(* IEC 61131-3 sources: beebread/doc (part 5) *)

(* ---- beedance_network.st ---- *)
// Commented out for beedance: it uses _STRING_TO_BUFFER, which is commented out.
// FUNCTION_BLOCK BASE64_DECODE_STR
// VAR_INPUT
// 	RUN : BOOL;
// END_VAR
// VAR_OUTPUT
// 	DONE : BOOL;
// END_VAR
// VAR_IN_OUT
// 	STR1 : STRING(192);
// 	STR2 : STRING(144);
// END_VAR
// VAR
// 	BASE64_DECODE_STREAM : BASE64_DECODE_STREAM;
// 	run_last : BOOL;
// 	buf1 : ARRAY [0..63] OF BYTE;
// 	buf2 : ARRAY [0..47] OF BYTE;
// 	mode : INT;
// 	size1 : INT;
// 	size2 : INT;
// 	end : INT;
// 	pos : INT;
// END_VAR
//
// CASE mode OF
// 0:	IF RUN AND NOT run_last THEN
// 		DONE := FALSE;
// 		mode := 1;
// 		end := LEN(STR1);
// 		pos := 0;
// 		STR2 := '';
// 	END_IF;
// 1:
// 	size1 := MIN(48,end - pos);
// 	IF size1 > 0 THEN
// 		_STRING_TO_BUFFER(STR:=MID(STR1, size1, pos + 1), POS:=0, PT:=REF(buf1), SIZE:=SIZEOF(buf1));
// 		BASE64_DECODE_STREAM(BUF1:=buf1 ,BUF2:=buf2 ,SIZE1:=size1 ,SIZE2=>size2);
// 		STR2 := CONCAT(STR2,BUFFER_TO_STRING(PT:=REF(buf2), SIZE:=SIZEOF(buf2), START:=0, STOP:=size2 - 1));
// 	ELSE
// 		mode := 0;
// 		DONE := TRUE;
// 	END_IF;
// 	pos := pos + size1;
// END_CASE;
//
// run_last := RUN;
// END_FUNCTION_BLOCK

FUNCTION_BLOCK BASE64_DECODE_STREAM
VAR_IN_OUT
	BUF1 : ARRAY [0..63] OF BYTE;
	BUF2 : ARRAY [0..47] OF BYTE;
END_VAR
VAR_INPUT
	SIZE1 : INT;
END_VAR
VAR_OUTPUT
	SIZE2 : INT;
END_VAR
VAR_TEMP
	a: INT;
	b: WORD;
	o: INT;
	off: INT;
	i1: INT;
	i2: INT;
	c: INT;
END_VAR

IF SIZE1 <= 0 THEN SIZE2 := 0; RETURN; END_IF;
c := SIZE1 - 1;
i2 := 0;
a := 0;
b := 0;
FOR i1 := 0 TO c DO
	o := BUF1[i1];
	IF o = 61 THEN (* = *)	EXIT;
	ELSIF o > 96 THEN (* a-z *) off := 71;
	ELSIF o > 64 THEN (* A-Z *) off := 65;
	ELSIF o > 47 THEN (* 0-9 *) off := -4;
	ELSIF o = 43 THEN (* + *) off := -19;
	ELSIF o = 47 THEN (* / *) off := -16;
	END_IF;
	b := SHL(b,6) OR INT_TO_BYTE(o - off);
	a := a + 6;
	IF a >= 8 THEN
		a := a - 8;
		BUF2[i2] := WORD_TO_BYTE(SHR(b,a));
		i2 := i2 + 1;
		b := b AND NOT SHL(WORD#16#FFFF,a);
	END_IF;
END_FOR;
SIZE2 := i2;
END_FUNCTION_BLOCK

// Commented out for beedance: it uses _STRING_TO_BUFFER, which is commented out.
// FUNCTION_BLOCK BASE64_ENCODE_STR
// VAR_INPUT
// 	RUN : BOOL;
// END_VAR
// VAR_OUTPUT
// 	DONE : BOOL;
// END_VAR
// VAR_IN_OUT
// 	STR1 : STRING(144);
// 	STR2 : STRING(192);
// END_VAR
// VAR
// 	BASE64_ENCODE_STREAM : BASE64_ENCODE_STREAM;
// 	run_last : BOOL;
// 	buf1 : ARRAY [0..47] OF BYTE;
// 	buf2 : ARRAY [0..63] OF BYTE;
// 	mode : INT;
// 	size1 : INT;
// 	size2 : INT;
// 	end : INT;
// 	pos : INT;
// END_VAR
//
// CASE mode OF
// 0:	IF RUN AND NOT run_last THEN
// 		DONE := FALSE;
// 		mode := 1;
// 		end := LEN(STR1);
// 		pos := 0;
// 		STR2 := '';
// 	END_IF;
// 1:
// 	size1 := MIN(48,end - pos);
// 	IF size1 > 0 THEN
// 		_STRING_TO_BUFFER(STR:=MID(STR1, size1, pos + 1), POS:=0, PT:=REF(buf1), SIZE:=SIZEOF(buf1));
// 		BASE64_ENCODE_STREAM(BUF1:=buf1 ,BUF2:=buf2 ,SIZE1:=size1 ,SIZE2=>size2);
// 		STR2 := CONCAT(STR2,BUFFER_TO_STRING(PT:=REF(buf2), SIZE:=SIZEOF(buf2), START:=0, STOP:=size2 - 1));
// 	ELSE
// 		mode := 0;
// 		DONE := TRUE;
// 	END_IF;
// 	pos := pos + size1;
// END_CASE;
//
// run_last := RUN;
// END_FUNCTION_BLOCK

// Commented out for beedance: it uses CODE, which is commented out.
// FUNCTION_BLOCK BASE64_ENCODE_STREAM
// VAR_IN_OUT
// 	BUF1 : ARRAY [0..47] OF BYTE;
// 	BUF2 : ARRAY [0..63] OF BYTE;
// END_VAR
// VAR_INPUT
// 	SIZE1 : INT;
// END_VAR
// VAR_OUTPUT
// 	SIZE2 : INT;
// END_VAR
// VAR
// 	a: INT;
// 	b: WORD;
// 	i: INT;
// 	i2: INT;
// 	i3: INT;
// 	c: INT;
// 	BASE64: STRING(64) := 'ABCDEFGHIJKLMNOPQRSTUVWXYZabcdefghijklmnopqrstuvwxyz0123456789+/';
// END_VAR
//
// IF SIZE1 <= 0 THEN
// 	SIZE2 := 0;
// 	RETURN;
// END_IF;
// c := SIZE1 - 1;
// i2 := 0;
// a := 0;
// b := 0;
// FOR i := 0 TO c DO
// 	b := SHL(b,8) OR BUF1[i];
// 	a := a + 8;
// 	WHILE a >= 6 DO
// 		a := a - 6;
// 		buf2[i2] := CODE(BASE64,WORD_TO_INT(SHR(b,a)) + 1);
// 		i2 := i2 + 1;
// 		b := b AND NOT SHL(WORD#16#FFFF,a);
// 	END_WHILE;
// END_FOR;
// IF a > 0 THEN
// 	buf2[i2] := CODE(BASE64,WORD_TO_INT(SHL(b,6 - a)) + 1);
// 	i2 := i2 + 1;
// 	i3 := i2 + (NOT INT_TO_WORD(i2) AND 2#11);
// 	FOR i := i2 TO i3 DO
// 		buf2[i] := 61;
// 	END_FOR;
// 	SIZE2 := i3 + 1;
// ELSE
// 	SIZE2 := i2;
// END_IF;
// END_FUNCTION_BLOCK

// Commented out for beedance: it reads or writes the bytes of a STRING through a pointer; a beedance reference (REF_TO) refers to a whole variable of its type.
// FUNCTION_BLOCK CSV_PARSER_BUF
// VAR_INPUT
// 	SEP : BYTE;
// END_VAR
// VAR_IN_OUT
// 	RUN : BYTE;
// 	OFFSET : UDINT;
// 	VALUE : STRING(STRING_LENGTH);
// 	PT : NETWORK_BUFFER;
// END_VAR
// VAR_OUTPUT
// 	RESULT : BYTE;
// END_VAR
// VAR
// 	step : INT;
// 	size : INT;
// 	c : BYTE;
// 	v_add : BYTE;
// 	i : INT;
// 	state : BYTE;
// 	eof : BOOL;
// 	pv : REF_TO BYTE;
// 	pve : DWORD;
// 	watchdog : TON;
// 	x : BOOL;
//
// 	(*LOG_MSG : LOG_MSG;
// 	_debug_enable : BOOL := TRUE;
// 	step_last : INT;*)
// END_VAR
//
// IF RUN > 0 THEN
// 	IF state = 0 THEN (* restart evaluation *)
//
// 		pv := REF(VALUE);
// 		pv^ := 0; (* VALUE = '' *)
// 		pve := pv + INT_TO_DWORD(STRING_LENGTH);
// 		i := UDINT_TO_INT(OFFSET);
// 		size := UINT_TO_INT(PT.SIZE) - 1;
// 		RESULT := 0;
// 		state := 5; (* command in progress (busy) *)
// 		step := 0; (* restart evaluation *)
//
// 		(* ---------------- Debug-Message -----------------------*)
// 		(*IF _debug_enable THEN
// 			LOG_CL.NEW_MSG := 'CPF: Startindex: ~1';
// 			LOG_CL.PRINTF[1] := INT_TO_STRING(i);
// 			LOG_MSG();
// 		END_IF;*)
// 		(* -----------------------------------------------------------------*)
//
// 	END_IF;
//
// 	watchdog(IN:=FALSE,PT:=T#1ms); (* restart timer *)
// 	watchdog.IN := TRUE;
//
// 	WHILE (state = 5) DO (* loop as long as there is no result *)
//
// 		watchdog(); (* update timer *)
//
// 		IF watchdog.Q THEN (* watchdog triggered *)
// 			state := 5;
// 			EXIT;
// 		ELSIF i > size THEN (* no further character available *)
// 			state := 10; (* nothing found - end of data reached *)
// 			EXIT;
// 		ELSE
//
// 			c := PT.BUFFER[i]; (* read new character from buffer *)
// 			eof := i + 1 = PT.SIZE; (* End of File *)
//
// 			v_add := 0;
//
// 			IF c = SEP THEN (* new element detected *)
// 				state := 1;
// 				x := TRUE;
// 			ELSIF c >= 32 THEN (* element detected *)
// 				v_add := c; (* store character *)
// 				IF eof THEN
// 					state := 2; (* element and end of line detected *)
// 				ELSE
// 					x := TRUE;
// 				END_IF;
// 			ELSE
// 				IF x THEN
// 					state := 2; (* element and end of line detected *)
// 					x := FALSE;
// 				END_IF;
// 			END_IF;
//
// 			IF v_add > 0  AND pv < pve THEN (* add character to value string *)
// 				pv^ := v_add; (* enter character *)
// 				pv := pv + 1;
// 				pv^ := 0; (* enter string termination *)
// 			END_IF;
//
// 			i := i + 1; (* increment data pointer *)
//
// 		END_IF;
// 	END_WHILE;
//
// 	CASE state OF
// 	01:	(* element found *)
// 		RESULT := 1; (* element found *)
// 		OFFSET := i; (* take offset *)
// 		RUN := 0;
// 		state := 0;
// 	02:	(* element found *)
// 		RESULT := 2; (* element and end of line detected *)
// 		OFFSET := i; (* take offset *)
// 		RUN := 0;
// 		state := 0;
//
// 	05:	RESULT := 5; (* in progress *)
//
// 	10:	(* index out of range - end of buffer *)
// 		RESULT := 10; (* nothing found - end of data reached *)
// 		OFFSET := i; (* take offset *)
// 		RUN := 0;
// 		state := 0;
// 	END_CASE;
//
// 	(* ---------------- Debug-Message -----------------------*)
// 	(*IF _debug_enable THEN
// 		LOG_CL.NEW_MSG := 'CPF: intern Result ~1 , state ~2, step ~3 , offset ~4, run ~5';
// 		LOG_CL.PRINTF[1] := BYTE_TO_STRING(RESULT);
// 		LOG_CL.PRINTF[2] := BYTE_TO_STRING(state);
// 		LOG_CL.PRINTF[3] := INT_TO_STRING(step);
// 		LOG_CL.PRINTF[4] := UDINT_TO_STRING(OFFSET);
// 		LOG_CL.PRINTF[5] := BYTE_TO_STRING(RUN);
// 		LOG_MSG();
// 	END_IF;*)
// 	(* -----------------------------------------------------------------*)
//
// END_IF;
//
// (* ---------------- Debug-Message -----------------------*)
// (*IF _debug_enable THEN
// 	IF step_last <> step THEN
// 		LOG_CL.NEW_MSG := 'IPB: Step: ~1';
// 		LOG_CL.PRINTF[1]  := INT_TO_STRING(step);
// 		LOG_MSG();
// 	END_IF;
// 	step_last := step;
// END_IF;*)
// (* -----------------------------------------------------------------*)
// END_FUNCTION_BLOCK

// Commented out for beedance: it reads or writes the bytes of a STRING through a pointer; a beedance reference (REF_TO) refers to a whole variable of its type.
// FUNCTION_BLOCK CSV_PARSER_FILE
// VAR_INPUT
// 	SEP : BYTE;
// END_VAR
// VAR_IN_OUT
// 	FILENAME : STRING;
// 	FSD : FILE_SERVER_DATA;
// 	RUN : BYTE;
// 	OFFSET : UDINT;
// 	VALUE : STRING(STRING_LENGTH);
// 	PT	: NETWORK_BUFFER;
// END_VAR
// VAR_OUTPUT
// 	RESULT : BYTE;
// END_VAR
// VAR
// 	i : UDINT;
// 	state : BYTE;
// 	e : BYTE;
// 	mode : BYTE;
// 	step : INT;
// 	c : BYTE;
// 	v_add : BYTE;
// 	eof : BOOL;
// 	pv : REF_TO BYTE;
// 	pve : DWORD;
// 	watchdog : TON;
// 	x : BOOL;
// 	FB : FILE_BLOCK;
//
// 	(*LOG_MSG : LOG_MSG;
// 	_debug_enable : BOOL := FALSE;
// 	step_last : INT;*)
// END_VAR
//
// IF RUN > 0 THEN
//
// 	IF state = 0 THEN (* restart evaluation *)
// 		pv := REF(VALUE);
// 		pv^ := 0; (* VALUE = '' *)
// 		pve := pv + INT_TO_DWORD(STRING_LENGTH);
// 		i := OFFSET;
// 		RESULT := 0;
// 		state := 5; (* command in progress (busy) *)
// 		step := 0; (* restart evaluation *)
//
// 		(* ---------------- Debug-Message -----------------------*)
// 		(*IF _debug_enable THEN
// 			LOG_CL.NEW_MSG := 'CPF: Startindex: ~1';
// 			LOG_CL.PRINTF[1] := UDINT_TO_STRING(i);
// 			LOG_MSG();
// 		END_IF;*)
// 		(* -----------------------------------------------------------------*)
//
// 	END_IF;
//
// 	watchdog(IN:=FALSE,PT:=T#1ms); (* restart timer *)
// 	watchdog.IN := TRUE;
//
// 	WHILE (state = 5) DO (* loop as long as there is no result *)
//
// 		mode := 1;
// 		FB(MODE:=mode,FSD:=fsd,PT:=PT,FILENAME:=FILENAME,POS:=i );
// 		e:=FB.ERROR;
// 		c:=FB.DATA;
//
// 		eof := i + 1 = FSD.FILE_SIZE; (* End of File *)
//
// 		(* ---------------- Debug-Message -----------------------*)
// 		(*IF _debug_enable THEN
// 			LOG_CL.NEW_MSG := 'CPF: mode: ~1, error: ~2 , >~7<>~3< ~4 step ~5 index ~6';
// 			LOG_CL.PRINTF[1] := BYTE_TO_STRING(mode);
// 			LOG_CL.PRINTF[2] := BYTE_TO_STRING(e);
// 			LOG_CL.PRINTF[3] := BYTE_TO_STRING(c);
// 			LOG_CL.PRINTF[4] := BOOL_TO_STRING(eof);
// 			LOG_CL.PRINTF[5] := INT_TO_STRING(step);
// 			LOG_CL.PRINTF[6] := UDINT_TO_STRING(i);
// 			LOG_CL.PRINTF[7] := CHR_TO_STRING(c);
// 			LOG_MSG();
// 		END_IF;*)
// 		(* -----------------------------------------------------------------*)
// 		watchdog(); (* update timer *)
//
// 		IF mode > 0 OR watchdog.Q THEN (* block still active, or watchdog triggered *)
// 			state := 5;
// 			EXIT;
// 		ELSIF e > 0 THEN (* File_error or no further character available *)
// 			state := 10; (* nothing found - end of data reached *)
// 			EXIT;
// 		ELSE
//
// 			v_add := 0;
//
// 			IF c = SEP THEN (* new element detected *)
// 				state := 1;
// 				x := TRUE;
// 			ELSIF c >= 32 THEN (* element detected *)
// 				v_add := c; (* store character *)
// 				IF eof THEN
// 					state := 2; (* element and end of line detected *)
// 				ELSE
// 					x := TRUE;
// 				END_IF;
// 			ELSE
// 				IF x THEN
// 					state := 2; (* element and end of line detected *)
// 					x := FALSE;
// 				END_IF;
// 			END_IF;
//
// 			IF v_add > 0  AND pv < pve THEN (* add character to value string *)
// 				pv^ := v_add; (* enter character *)
// 				pv := pv + 1;
// 				pv^ := 0; (* enter string termination *)
// 			END_IF;
//
// 			i := i + 1; (* increment data pointer *)
//
// 		END_IF;
// 	END_WHILE;
//
// 	CASE state OF
// 	01:	(* element found *)
// 		RESULT := 1; (* element found *)
// 		OFFSET := i; (* take offset *)
// 		RUN := 0;
// 		state := 0;
// 	02:	(* element found *)
// 		RESULT := 2; (* element and end of line detected *)
// 		OFFSET := i; (* take offset *)
// 		RUN := 0;
// 		state := 0;
//
// 	05:	RESULT := 5; (* in progress *)
//
// 	10:	(* index out of range - end of buffer *)
// 		RESULT := 10; (* nothing found - end of data reached *)
// 		OFFSET := i; (* take offset *)
// 		RUN := 0;
// 		state := 0;
// 	END_CASE;
//
// 	(* ---------------- Debug-Message -----------------------*)
// 	(*IF _debug_enable THEN
// 		LOG_CL.NEW_MSG := 'CPF: intern Result ~1 , state ~2, step ~3 , offset ~4, run ~5';
// 		LOG_CL.PRINTF[1] := BYTE_TO_STRING(RESULT);
// 		LOG_CL.PRINTF[2] := BYTE_TO_STRING(state);
// 		LOG_CL.PRINTF[3] := INT_TO_STRING(step);
// 		LOG_CL.PRINTF[4] := UDINT_TO_STRING(OFFSET);
// 		LOG_CL.PRINTF[5] := BYTE_TO_STRING(RUN);
// 		LOG_MSG();
// 	END_IF;*)
// 	(* -----------------------------------------------------------------*)
//
// END_IF;
//
// (* ---------------- Debug-Message -----------------------*)
// (*IF _debug_enable THEN
// 	IF step_last <> step THEN
// 		LOG_CL.NEW_MSG := 'CPF: Step: ~1';
// 		LOG_CL.PRINTF[1]  := INT_TO_STRING(step);
// 		LOG_MSG();
// 	END_IF;
// 	step_last := step;
// END_IF;*)
// (* -----------------------------------------------------------------*)
// END_FUNCTION_BLOCK

// Commented out for beedance: it uses UNI_CIRCULAR_BUFFER, which is commented out.
// FUNCTION_BLOCK DLOG_BOOL
// VAR_IN_OUT
// 	X : DLOG_DATA;
// END_VAR
// VAR_INPUT
// 	STATE : BOOL;
// 	OFF : STRING;
// 	ON : STRING;
// 	COLUMN : STRING(40);
// 	DELTA : BOOL;
// END_VAR
// VAR_OUTPUT
// END_VAR
// VAR
// 	UCB : UNI_CIRCULAR_BUFFER;
// 	id : WORD;
// 	last_delta : BOOL;
// 	state_last: BOOL;
// END_VAR
//
// CASE x.ADD_COM OF
//
// 01:	(* ADD INFO *)
// 	X.ID_MAX := X.ID_MAX + USINT#1;
// 	id := WORD#16#0601; (* source type BOOL, target type STRING *)
// 02:	(* ADD HEADER *)
// 	X.UCB.D_STRING := COLUMN;
// 	X.UCB.D_HEAD := id;
// 	X.UCB.D_MODE := 1;
// 	UCB(DATA:=X.UCB); (* enter data *)
// 03:	(* ADD DATA *)
// 	IF X.STORE_TYPE = BYTE#05 THEN (* MySQL mode *)
// 		X.UCB.D_STRING := SEL(state_last,'0','1');
// 	ELSE
// 		X.UCB.D_STRING := SEL(state_last,OFF,ON);
// 	END_IF;
// 	X.UCB.D_HEAD := id;
//
// 	X.UCB.D_MODE := 1;
// 	UCB(DATA:=X.UCB); (* enter data *)
// 	last_delta := STATE;
// 04:	(* ADD DATA REQ *)
// 	IF DELTA AND (STATE XOR last_delta) THEN
// 		X.ADD_DATA_REQ := TRUE;
// 		last_delta := STATE;
// 	END_IF;
// END_CASE;
// state_last := STATE;
// END_FUNCTION_BLOCK

// Commented out for beedance: it uses ELEMENT_GET, which is commented out.
// FUNCTION_BLOCK DLOG_CRON_TAB
// VAR_INPUT
// 	ACTIVATE : BOOL;
// 	DTI : DT;
// 	SECOND : STRING(20);
// 	MINUTE : STRING(20);
// 	HOUR : STRING(20);
// 	DAY_OF_MONTH : STRING(20);
// 	DAY_OF_WEEK : STRING(20);
// 	MONTH : STRING(20);
// END_VAR
// VAR_OUTPUT
// 	Q : BOOL;
// END_VAR
// VAR
// 	CD :  DLOG_CRON_DATA;
// 	activate_old : BOOL;
// 	datei : DATE;
// 	dti_last : DT;
// 	cnt1 : INT;
// 	cnt2 : INT;
// 	idx1 : INT;
// 	idx2 : INT;
// 	idx3 : INT;
// 	idx4 : INT;
// 	pos1 : INT;
// 	pos2 : INT;
// 	char_cnt : INT;
// 	trig_day : BOOL;
// 	trig_weekday : BOOL;
// 	str1 : STRING(STRING_LENGTH);
// 	str2 : STRING(STRING_LENGTH);
// 	str3 : STRING(STRING_LENGTH);
// 	num_str1 : STRING(10);
// END_VAR
//
// IF ACTIVATE THEN
// 	IF NOT activate_old THEN
// 		CD.CE[0].VALUE_MIN := 0;	(* seconds *)
// 		CD.CE[0].VALUE_MAX := 59;
// 		CD.CE[1].VALUE_MIN := 0;	(* minutes *)
// 		CD.CE[1].VALUE_MAX := 59;
// 		CD.CE[2].VALUE_MIN := 0;	(* hours *)
// 		CD.CE[2].VALUE_MAX := 59;
// 		CD.CE[3].VALUE_MIN := 1;	(* days *)
// 		CD.CE[3].VALUE_MAX := 31;
// 		CD.CE[4].VALUE_MIN := 1;	(* weekday *)
// 		CD.CE[4].VALUE_MAX := 7;
// 		CD.CE[5].VALUE_MIN := 1;	(* month *)
// 		CD.CE[5].VALUE_MAX := 12;
//
// 		FOR idx1 := 0 TO 5 DO
// 			idx3 := CD.CE[idx1].VALUE_MIN;
// 			idx4 := CD.CE[idx1].VALUE_MAx;
// 			FOR idx2 := idx3 TO idx4 DO
// 				CD.CE[idx1].ELEMENTS[idx2] := FALSE;
// 			END_FOR;
// 			CD.CE[idx1].ALL_SELECTED := FALSE;
// 		END_FOR;
//
// 		str1 := CONCAT(SECOND,'#');
// 		str1 := CONCAT(str1,MINUTE);
// 		str1 := CONCAT(str1,'#');
// 		str1 := CONCAT(str1,HOUR);
// 		str1 := CONCAT(str1,'#');
// 		str1 := CONCAT(str1,DAY_OF_MONTH);
// 		str1 := CONCAT(str1,'#');
// 		str1 := CONCAT(str1,DAY_OF_WEEK);
// 		str1 := CONCAT(str1,'#');
// 		str1 := CONCAT(str1,MONTH);
//
// 		FOR idx1 := 0 TO 5 DO
// 			str2 := ELEMENT_GET(BYTE#35, idx1, str1);
// 			IF LEN(str2) > 0 THEN
// 				cnt1 := ELEMENT_COUNT(BYTE#44, str2);	(* separator ',' *)
// 			ELSE
// 				cnt1 := 1;
// 			END_IF;
//
// 			FOR idx2 := 0 TO cnt1 -1 DO
// 				str3 := ELEMENT_GET(BYTE#44, idx2, str2);
// 				IF FIND(str3, '*/') > 0 AND LEN(str3) <= 10 THEN
// 					pos1 := DEC_TO_INT(str3);
// 					IF pos1 > 0 THEN
// 						idx3 := CD.CE[idx1].VALUE_MIN;
// 						idx4 := CD.CE[idx1].VALUE_MAX;
// 						WHILE idx3 <= idx4 DO
// 							CD.CE[idx1].ELEMENTS[idx3] := TRUE;
// 							idx3 := idx3 + pos1;
// 						END_WHILE;
// 					END_IF;
//
// 				ELSE
// 					IF FIND(str3, '*') > 0 OR LEN(str3) = 0 THEN
// 						pos1 := CD.CE[idx1].VALUE_MIN;
// 						pos2 := CD.CE[idx1].VALUE_MAX;
// 						CD.CE[idx1].ALL_SELECTED := TRUE;
// 					ELSE
// 						cnt2 := ELEMENT_COUNT(BYTE#45, str3);	(* separator '-' *)
// 						char_cnt := LEN(str3);
// 						IF char_cnt >= 1 AND char_cnt <= 10 THEN
// 							num_str1 := ELEMENT_GET(BYTE#45, 0, str3);
// 							pos1 := DEC_TO_INT(num_str1);
// 							pos2 := pos1;
// 							IF cnt2 = 2 THEN
// 								num_str1 := ELEMENT_GET(BYTE#45, 1, str3);
// 								pos2 := DEC_TO_INT(num_str1);
// 							END_IF;
// 						END_IF;
// 					END_IF;
//
// 					IF pos1 >= CD.CE[idx1].VALUE_MIN AND pos2 <= CD.CE[idx1].VALUE_MAX THEN
// 						FOR idx3 := pos1 TO pos2 DO
// 							CD.CE[idx1].ELEMENTS[idx3] := TRUE;
// 						END_FOR;
// 					END_IF;
// 				END_IF;
// 			END_FOR;
// 		END_FOR;
// 	ELSIF DTI <> dti_last THEN
// 		CD.CE[0].VALUE := SECOND_OF_DT(DTI); (* seconds *)
// 		CD.CE[1].VALUE := MINUTE_OF_DT(DTI); (* minutes *)
// 		CD.CE[2].VALUE := HOUR_OF_DT(DTI); (* hours *)
// 		datei := DT_TO_DATE(DTI);
// 		CD.CE[3].VALUE := DAY_OF_MONTH(datei); (* Tag *)
// 		CD.CE[4].VALUE := DAY_OF_WEEK(datei); (* weekday *)
// 		CD.CE[5].VALUE := MONTH_OF_DATE(datei); (*  month *)
// 		dti_last := DTI;
//
// 		idx2 := CD.CE[0].VALUE;	(* seconds *)
// 		Q := CD.CE[0].ELEMENTS[idx2] = TRUE;
// 		idx2 := CD.CE[1].VALUE;	(* minutes *)
// 		Q := Q AND CD.CE[1].ELEMENTS[idx2] = TRUE;
// 		idx2 := CD.CE[2].VALUE;	(* hours *)
// 		Q := Q AND CD.CE[2].ELEMENTS[idx2] = TRUE;
// 		idx2 := CD.CE[5].VALUE;	(* month *)
// 		Q := Q AND CD.CE[5].ELEMENTS[idx2] = TRUE;
//
// 		(* evaluate day and weekday *)
// 		idx2 := CD.CE[3].VALUE;	(* Tag *)
// 		trig_day:= CD.CE[3].ELEMENTS[idx2] = TRUE;
// 		idx2 := CD.CE[4].VALUE;	(* weekday *)
// 		trig_weekday := CD.CE[4].ELEMENTS[idx2] = TRUE;
//
// 		IF CD.CE[3].ALL_SELECTED = FALSE AND CD.CE[4].ALL_SELECTED = TRUE THEN
// 			Q := Q AND trig_day; (* evaluate day only *)
// 		ELSIF CD.CE[3].ALL_SELECTED = TRUE AND CD.CE[4].ALL_SELECTED = FALSE THEN
// 			Q := Q AND trig_weekday; (* evaluate weekday only *)
// 		ELSIF CD.CE[3].ALL_SELECTED = FALSE AND CD.CE[4].ALL_SELECTED = FALSE THEN
// 			Q := Q AND (trig_weekday OR trig_day); (* evaluate day and weekday *)
// 		END_IF;
// 	END_IF;
//
// END_IF;
// activate_old := ACTIVATE;
// END_FUNCTION_BLOCK

// Commented out for beedance: it uses UNI_CIRCULAR_BUFFER, which is commented out.
// FUNCTION_BLOCK DLOG_DINT
// VAR_IN_OUT
// 	X : DLOG_DATA;
// END_VAR
// VAR_INPUT
// 	VALUE : DINT;
// 	COLUMN : STRING(40);
// 	DELTA : DINT;
// END_VAR
// VAR
// 	UCB : UNI_CIRCULAR_BUFFER;
// 	id : WORD;
// 	delta_last : DINT;
// 	value_last : DINT;
// END_VAR
//
// CASE x.ADD_COM OF
//
// 01:	(* ADD INFO *)
// 	X.ID_MAX := X.ID_MAX + USINT#1;
// 	id := WORD#16#0801; (* source type DINT, target type STRING *)
// 02:	(* ADD HEADER *)
// 	X.UCB.D_STRING := COLUMN;
// 	X.UCB.D_HEAD := id;
// 	X.UCB.D_MODE := 1;
// 	UCB(DATA:=X.UCB); (* enter data *)
// 03:	(* ADD DATA *)
// 	X.UCB.D_STRING := DINT_TO_STRING(value_last);
// 	X.UCB.D_HEAD := id;
// 	X.UCB.D_MODE := 1;
// 	UCB(DATA:=X.UCB); (* enter data *)
// 	delta_last := value_last;
// 04:	(* ADD DATA REQ *)
// 	IF DELTA <> DINT#0 THEN
// 		IF VALUE <= (delta_last - DELTA) OR VALUE >= (delta_last + DELTA) THEN
// 			X.ADD_DATA_REQ := TRUE;
// 			delta_last := VALUE;
// 		END_IF;
// 	END_IF;
// END_CASE;
// value_last := VALUE;
// END_FUNCTION_BLOCK

// Commented out for beedance: it uses UNI_CIRCULAR_BUFFER, which is commented out.
// FUNCTION_BLOCK DLOG_DT
// VAR_IN_OUT
// 	X : DLOG_DATA;
// END_VAR
// VAR_INPUT
// 	FMT : STRING := '#A-#D-#H #N:#R:#T';
// 	COLUMN : STRING(40);
// 	DELTA : UDINT;
// END_VAR
//
// VAR_OUTPUT
// END_VAR
// VAR
// 	UCB : UNI_CIRCULAR_BUFFER;
// 	id : WORD;
// 	delta_last : DT;
// END_VAR
//
// CASE x.ADD_COM OF
//
// 01:	(* ADD INFO *)
// 	X.ID_MAX := X.ID_MAX + USINT#1;
// 	id := WORD#16#0D01; (* source type DT, target type STRING *)
// 02:	(* ADD HEADER *)
// 	X.UCB.D_STRING := COLUMN;
// 	X.UCB.D_HEAD := id;
// 	X.UCB.D_MODE := 1;
// 	UCB(DATA:=X.UCB); (* enter data *)
// 03:	(* ADD DATA *)
// 	X.UCB.D_STRING := DT_TO_STRF(DTI:=X.DTI,MS:=0,FMT:=FMT,LANG:=0);
// 	X.UCB.D_HEAD := id;
// 	X.UCB.D_MODE := 1;
// 	UCB(DATA:=X.UCB); (* enter data *)
// 	delta_last := X.DTI;
// 04:	(* ADD DATA REQ *)
// 	IF DELTA <> UDINT#0 THEN
// 		IF DT_TO_UDINT(X.DTI) >= (DT_TO_UDINT(delta_last) + DELTA) THEN
// 			X.ADD_DATA_REQ := TRUE;
// 			delta_last := X.DTI;
// 		END_IF;
// 	END_IF;
// END_CASE;
// END_FUNCTION_BLOCK

// Commented out for beedance: it uses UNI_CIRCULAR_BUFFER, which is commented out.
// FUNCTION_BLOCK DLOG_FILE_TO_FTP
// VAR_IN_OUT
// 	X : DLOG_DATA;
// END_VAR
// VAR_INPUT
// 	FTP_URL : STRING(STRING_LENGTH);
// 	FTP_ACTIV : BOOL;
// 	FILE_DELETE : BOOL;
// 	TIMEOUT : TIME := T#30s;
// 	RETRY : INT;
// 	RETRY_TIME : TIME := T#30s;
// 	DNS_IP4 : DWORD;
// 	PLC_IP4 : DWORD;
// END_VAR
// VAR_OUTPUT
// 	DONE : BOOL;
// 	BUSY : BOOL;
// 	ERROR_C : DWORD;
// 	ERROR_T : BYTE;
// END_VAR
// VAR
// 	UCBD : UNI_CIRCULAR_BUFFER_DATA;
// 	UCB : UNI_CIRCULAR_BUFFER;
// 	FTP_CLIENT : FTP_CLIENT;
// 	WT_1 : TON;
// 	ftrig_old : BOOL;
// 	filename : STRING;
// 	step : INT;
// 	ftp_busy : BOOL;
// 	ftp_done : BOOL;
// 	cnt : INT;
//
// 	(*LOG_MSG : LOG_MSG;
// 	_debug_enable : BOOL := TRUE;*)
// END_VAR
//
// (* store new file name *)
// IF X.NEW_FILE_RTRIG AND ftrig_old = FALSE THEN
// 	UCBD.D_HEAD := 1;
// 	UCBD.D_MODE := 1;
// 	UCBD.D_STRING := X.NEW_FILE;
// 	UCB(DATA:=UCBD); (* enter data *)
// END_IF;
// ftrig_old := X.NEW_FILE_RTRIG;
//
// CASE step OF
//
// 00:	IF UCBD.BUF_COUNT > 0 AND ftp_busy = FALSE THEN
// 		UCBD.D_MODE := 12; (* read and delete data *)
// 		UCB(DATA:=UCBD);
// 		filename := UCBD.D_STRING;
// 		cnt := RETRY;
// 		step := 10;
//
// 		(*####################  DEBUG-MESSAGE  ###################################*)
// 		(*IF _debug_enable THEN
// 			LOG_CL.NEW_MSG := 'F_T_FTP: Auftrag aktiv /file: ~2';
// 			LOG_CL.PRINTF[2] := files;
// 			LOG_MSG();
// 		END_IF;*)
// 		(*########################################################################*)
//
// 	END_IF;
//
// 10:	IF ftp_busy = FALSE THEN
// 		IF ftp_done THEN
// 			(*####################  DEBUG-MESSAGE  ###################################*)
// 			(*IF _debug_enable THEN
// 				LOG_CL.NEW_MSG := 'F_T_FTP: Auftrag OK /file: ~2';
// 				LOG_CL.PRINTF[2] := filename;
// 				LOG_MSG();
// 			END_IF;*)
// 			(*########################################################################*)
// 			step := 0;
// 		ELSE
// 			step := 20; (* pause after error *)
// 		END_IF;
// 	END_IF;
//
// 20:	IF WT_1.Q THEN (* wait time *)
// 		cnt := cnt - 1;
// 		IF RETRY = 0 THEN (* repeat FTP transfer indefinitely *)
// 			(*####################  DEBUG-MESSAGE  ###################################*)
// 			(*IF _debug_enable THEN
// 				LOG_CL.NEW_MSG := 'F_T_FTP: Auftrag unbegrenzt wiederholen /file: ~2';
// 				LOG_CL.PRINTF[2] := filename;
// 				LOG_MSG();
// 			END_IF;*)
// 			(*########################################################################*)
// 			step := 10; (* repeat FTP transfer *)
// 		ELSIF cnt >= 0 THEN
// 			(*####################  DEBUG-MESSAGE  ###################################*)
// 			(*IF _debug_enable THEN
// 				LOG_CL.NEW_MSG := 'F_T_FTP: Auftrag wiederholen /cnt: ~1 /file: ~2';
// 				LOG_CL.PRINTF[1] := INT_TO_STRING(cnt);
// 				LOG_CL.PRINTF[2] := filename;
// 				LOG_MSG();
// 			END_IF;*)
// 			(*########################################################################*)
// 			step := 10; (* repeat FTP transfer *)
// 		ELSE
// 			(*####################  DEBUG-MESSAGE  ###################################*)
// 			(*IF _debug_enable THEN
// 				LOG_CL.NEW_MSG := 'F_T_FTP: Auftrag verworfen /file: ~2';
// 				LOG_CL.PRINTF[2] := filename;
// 				LOG_MSG();
// 			END_IF;*)
// 			(*########################################################################*)
// 			step := 0; (* discard FTP job *)
// 		END_IF;
// 	END_IF;
//
// END_CASE;
//
// BUSY := step = 10;
// DONE := step = 0;
// WT_1(IN:= step = 20, PT:= RETRY_TIME);
//
// FTP_CLIENT(
// 	ACTIVATE:= BUSY,
// 	FILENAME:= filename,
// 	FTP_URL:= FTP_URL,
// 	FTP_DOWNLOAD:= FALSE,
// 	FTP_ACTIV:= FTP_ACTIV,
// 	FILE_DELETE:= FILE_DELETE,
// 	TIMEOUT:= TIMEOUT,
// 	DNS_IP4:= DNS_IP4,
// 	PLC_IP4:= PLC_IP4,
// 	DONE=> ftp_done,
// 	BUSY=> ftp_busy
// 	);
//
// (* error evaluation *)
// IF FTP_CLIENT.ERROR_T <> BYTE#0 THEN
// 	ERROR_C := FTP_CLIENT.ERROR_C;
// 	ERROR_T := FTP_CLIENT.ERROR_T;
// ELSIF UCBD.BUF_DATA_LOST > UDINT#0 THEN
// 	ERROR_C := DWORD#2; (* error: buffer overflow - reduce amount of data *)
// 	ERROR_T := BYTE#6; 	(* Type: Buffer *)
// ELSIF UCBD.BUF_USED_MAX > USINT#90 THEN
// 	ERROR_C := DWORD#1; (* warning: buffer utilization > 90% *)
// 	ERROR_T := BYTE#6;	(* Type: Buffer *)
// ELSE
// 	ERROR_C := DWORD#0;
// 	ERROR_T := BYTE#0;
// END_IF;
// END_FUNCTION_BLOCK

// Commented out for beedance: it uses UNI_CIRCULAR_BUFFER, which is commented out.
// FUNCTION_BLOCK DLOG_FILE_TO_SMTP
// VAR_IN_OUT
// 	SERVER : STRING;
// 	MAILFROM : STRING;
// 	MAILTO : STRING(STRING_LENGTH);
// 	SUBJECT : STRING;
// 	BODY : STRING(STRING_LENGTH);
// 	X : DLOG_DATA;
// END_VAR
// VAR_INPUT
// 	FILE_DELETE : BOOL;
// 	TIMEOUT : TIME := T#30s;
// 	DTI : DT;
// 	DTI_OFFSET : INT;
// 	RETRY : INT;
// 	RETRY_TIME : TIME := T#30s;
// 	DNS_IP4 : DWORD;
// END_VAR
// VAR_OUTPUT
// 	DONE : BOOL;
// 	BUSY : BOOL;
// 	ERROR_C : DWORD;
// 	ERROR_T : BYTE;
// END_VAR
// VAR
// 	UCBD : UNI_CIRCULAR_BUFFER_DATA;
// 	UCB : UNI_CIRCULAR_BUFFER;
// 	SMTP_CLIENT : SMTP_CLIENT;
// 	WT_1 : TON;
// 	ftrig_old : BOOL;
// 	files : STRING(STRING_LENGTH);
// 	step : INT;
// 	smtp_busy : BOOL;
// 	smtp_done : BOOL;
// 	cnt : INT;
//
// 	(*LOG_MSG : LOG_MSG;
// 	_debug_enable : BOOL := TRUE;*)
// END_VAR
//
// (* store new file name *)
// IF X.NEW_FILE_RTRIG AND ftrig_old = FALSE THEN
// 	UCBD.D_HEAD := 1;
// 	UCBD.D_MODE := 1;
// 	UCBD.D_STRING := X.NEW_FILE;
// 	UCB(DATA:=UCBD); (* enter data *)
// END_IF;
// ftrig_old := X.NEW_FILE_RTRIG;
//
// CASE step OF
//
// 00:	IF UCBD.BUF_COUNT > 0 AND smtp_busy = FALSE THEN
// 		UCBD.D_MODE := 12; (* read and delete data *)
// 		UCB(DATA:=UCBD);
// 		files := UCBD.D_STRING;
// 		IF FILE_DELETE THEN
// 			files := CONCAT(files,';#DEL#');
// 		END_IF;
// 		cnt := RETRY;
// 		step := 10;
//
// 		(*####################  DEBUG-MESSAGE  ###################################*)
// 		(*IF _debug_enable THEN
// 			LOG_CL.NEW_MSG := 'F_T_SMTP: Auftrag aktiv /file: ~2';
// 			LOG_CL.PRINTF[2] := files;
// 			LOG_MSG();
// 		END_IF;*)
// 		(*########################################################################*)
//
// 	END_IF;
//
// 10:	IF smtp_busy = FALSE THEN
// 		IF smtp_done THEN
// 			(*####################  DEBUG-MESSAGE  ###################################*)
// 			(*IF _debug_enable THEN
// 				LOG_CL.NEW_MSG := 'F_T_SMTP: Auftrag OK /file: ~2';
// 				LOG_CL.PRINTF[2] := files;
// 				LOG_MSG();
// 			END_IF;*)
// 			(*########################################################################*)
// 			step := 0;
// 		ELSE
// 			step := 20; (* pause after error *)
// 		END_IF;
// 	END_IF;
//
// 20:	IF WT_1.Q THEN (* wait time *)
// 		cnt := cnt - 1;
// 		IF RETRY = 0 THEN (* repeat transfer indefinitely *)
// 			(*####################  DEBUG-MESSAGE  ###################################*)
// 			(*IF _debug_enable THEN
// 				LOG_CL.NEW_MSG := 'F_T_SMTP: Auftrag unbegrenzt wiederholen /file: ~2';
// 				LOG_CL.PRINTF[2] := files;
// 				LOG_MSG();
// 			END_IF;*)
// 			(*########################################################################*)
// 			step := 10; (* repeat transfer *)
// 		ELSIF cnt >= 0 THEN
// 			(*####################  DEBUG-MESSAGE  ###################################*)
// 			(*IF _debug_enable THEN
// 				LOG_CL.NEW_MSG := 'F_T_SMTP: Auftrag wiederholen /cnt: ~1 /file: ~2';
// 				LOG_CL.PRINTF[1] := INT_TO_STRING(cnt);
// 				LOG_CL.PRINTF[2] := files;
// 				LOG_MSG();
// 			END_IF;*)
// 			(*########################################################################*)
// 			step := 10; (* repeat transfer *)
// 		ELSE
// 			(*####################  DEBUG-MESSAGE  ###################################*)
// 			(*IF _debug_enable THEN
// 				LOG_CL.NEW_MSG := 'F_T_SMTP: Auftrag verworfen /file: ~2';
// 				LOG_CL.PRINTF[2] := files;
// 				LOG_MSG();
// 			END_IF;*)
// 			(*########################################################################*)
// 			step := 0; (* discard job *)
// 		END_IF;
// 	END_IF;
//
// END_CASE;
//
// BUSY := step = 10;
// DONE := step = 0;
// WT_1(IN:= step = 20, PT:= RETRY_TIME);
//
// SMTP_CLIENT(
// 	ACTIVATE:= BUSY,
// 	TIMEOUT:= TIMEOUT,
// 	DTI:= DTI,
// 	DTI_OFFSET:= DTI_OFFSET,
// 	DNS_IP4:= DNS_IP4,
// 	SERVER:= SERVER,
// 	MAILFROM:= MAILFROM,
// 	MAILTO:= MAILTO,
// 	SUBJECT:= SUBJECT,
// 	BODY:= BODY,
// 	FILES:= FILES,
// 	DONE=> smtp_done,
// 	BUSY=> smtp_busy
// 	);
//
// (* error evaluation *)
// IF SMTP_CLIENT.ERROR_T <> BYTE#0 THEN
// 	ERROR_C := SMTP_CLIENT.ERROR_C;
// 	ERROR_T := SMTP_CLIENT.ERROR_T;
// ELSIF UCBD.BUF_DATA_LOST > UDINT#0 THEN
// 	ERROR_C := DWORD#2; (* error: buffer overflow - reduce amount of data *)
// 	ERROR_T := BYTE#6; 	(* Type: Buffer *)
// ELSIF UCBD.BUF_USED_MAX > USINT#90 THEN
// 	ERROR_C := DWORD#1; (* warning: buffer utilization > 90% *)
// 	ERROR_T := BYTE#6;	(* Type: Buffer *)
// ELSE
// 	ERROR_C := DWORD#0;
// 	ERROR_T := BYTE#0;
// END_IF;
// END_FUNCTION_BLOCK

// Commented out for beedance: it uses UNI_CIRCULAR_BUFFER, which is commented out.
// FUNCTION_BLOCK DLOG_REAL
// VAR_IN_OUT
// 	X : DLOG_DATA;
// END_VAR
// VAR_INPUT
// 	VALUE : REAL;
// 	N : INT;
// 	D : STRING(1) := ',';
// 	COLUMN : STRING(40);
// 	DELTA : REAL;
// END_VAR
// VAR
// 	UCB : UNI_CIRCULAR_BUFFER;
// 	id : WORD;
// 	delta_last : REAL;
// 	value_last : REAL;
// END_VAR
//
// CASE x.ADD_COM OF
//
// 01:	(* ADD INFO *)
// 	X.ID_MAX := X.ID_MAX + USINT#1;
// 	id := WORD#16#0201; (* source type REAL, target type STRING *)
// 02:	(* ADD HEADER *)
// 	X.UCB.D_STRING := COLUMN;
// 	X.UCB.D_HEAD := id;
// 	X.UCB.D_MODE := 1;
// 	UCB(DATA:=X.UCB); (* enter data *)
// 03:	(* ADD DATA *)
// 	X.UCB.D_STRING := REAL_TO_STRF(IN:=value_last,N:=N,D:=D);
// 	X.UCB.D_HEAD := id;
// 	X.UCB.D_MODE := 1;
// 	UCB(DATA:=X.UCB); (* enter data *)
// 	delta_last := value_last;
// 04:	(* ADD DATA REQ *)
// 	IF DELTA <> 0.0 THEN
// 		IF VALUE <= (delta_last - DELTA) OR VALUE >= (delta_last + DELTA) THEN
// 			X.ADD_DATA_REQ := TRUE;
// 			delta_last := VALUE;
// 		END_IF;
// 	END_IF;
// END_CASE;
// value_last := VALUE;
// END_FUNCTION_BLOCK

// Commented out for beedance: it uses UNI_CIRCULAR_BUFFER, which is commented out.
// FUNCTION_BLOCK DLOG_REAL_ARRAY
// VAR_IN_OUT
// 	R_ARRAY : DLOG_REAL_ARRAY_DATA;
// 	X : DLOG_DATA;
// END_VAR
// VAR_INPUT
// 	N : INT;
// 	D : STRING(1);
// 	R_COUNT : INT;
// END_VAR
// VAR
// 	UCB : UNI_CIRCULAR_BUFFER;
// 	id : WORD;
// 	idx : INT;
// END_VAR
//
// FOR idx := 1 TO R_COUNT DO
//
// 	CASE x.ADD_COM OF
//
// 	01:	(* ADD INFO *)
// 		X.ID_MAX := X.ID_MAX + USINT#1;
// 		id := WORD#16#0201; (* source type REAL, target type STRING *)
// 		(* assign name automatically *)
// 		IF LEN(R_ARRAY[idx].COLUMN) = 0 THEN
// 			R_ARRAY[idx].COLUMN := CONCAT('Spalte_',USINT_TO_STRING(X.ID_MAX));
// 		END_IF;
// 	02:	(* ADD HEADER *)
// 		X.UCB.D_STRING := R_ARRAY[idx].COLUMN;
// 		X.UCB.D_HEAD := id;
// 		X.UCB.D_MODE := 1;
// 		UCB(DATA:=X.UCB); (* enter data *)
// 	03:	(* ADD DATA *)
// 		X.UCB.D_STRING := REAL_TO_STRF(IN:=R_ARRAY[idx]._value_last,N:=N,D:=D);
// 		X.UCB.D_HEAD := id;
// 		X.UCB.D_MODE := 1;
// 		UCB(DATA:=X.UCB); (* enter data *)
// 		R_ARRAY[idx]._delta_last := R_ARRAY[idx]._value_last;
// 	04:	(* ADD DATA REQ *)
// 		IF R_ARRAY[idx].DELTA <> 0.0 THEN
// 			IF R_ARRAY[idx].VALUE <= (R_ARRAY[idx]._delta_last - R_ARRAY[idx].DELTA) OR R_ARRAY[idx].VALUE >= (R_ARRAY[idx]._delta_last + R_ARRAY[idx].DELTA) THEN
// 				X.ADD_DATA_REQ := TRUE;
// 				R_ARRAY[idx]._delta_last := R_ARRAY[idx].VALUE;
// 			END_IF;
// 		END_IF;
// 	END_CASE;
// 	R_ARRAY[idx]._value_last := R_ARRAY[idx].VALUE;
//
// END_FOR;
// END_FUNCTION_BLOCK

// Commented out for beedance: it names a variable fn, which beedance reads as its function keyword.
// FUNCTION_BLOCK DLOG_STORE_FILE_CSV
// VAR_IN_OUT
// 	X : DLOG_DATA;
// 	SAVE_DATA : DLOG_SAVE;
// END_VAR
// VAR_INPUT
// 	ENABLE : BOOL;
// 	TRIG_M : BOOL;
// 	TRIG_T : TIME;
// 	FILENAME : STRING;
// 	DTI : DT;
// 	SEP : BYTE;
// 	AUTO_CLOSE : TIME := T#15s;
// END_VAR
// VAR_OUTPUT
// 	ERROR_C : DWORD;
// 	ERROR_T : BYTE;
// END_VAR
// VAR
// 	FS : FILE_SERVER;
// 	FSD : FILE_SERVER_DATA;
// 	PT : NETWORK_BUFFER;
// 	UCB : UNI_CIRCULAR_BUFFER;
// 	trig_auto : BOOL;
// 	trig_stored : BOOL;
// 	trig_tmp : BOOL;
// 	trig_m_last : BOOL;
// 	dti_last : DT := DT#2070-02-06-06:28:15;
// 	fn_last : STRING;
// 	fn : STRING;
// 	step_1: INT;
// 	step_2: INT;
// 	idx : INT;
// 	log_stop : BOOL;
// 	n : USINT;
// 	wd_ton : TON;
// 	wd_time : TIME;
// 	aw_ton : TON;
// 	aw_enable : BOOL;
// 	aw_aktiv : BOOL;
// 	total_bytes : UDINT;
//
// 	(*
// 	LOG_MSG : LOG_MSG;
// 	_debug_enable : BOOL := TRUE;
// 	*)
// END_VAR
//
// X.DTI := DTI; (* enter date / time *)
// X.CLOCK_TRIG := DTI <> dti_last;
// dti_last := DTI;
// trig_auto := FALSE;
// IF X.CLOCK_TRIG THEN (* pulse every second *)
// 	fn := DT_TO_STRF(DTI, 0, FILENAME, 0); (* automatic file name generation *)
// 	IF TRIG_T >= T#1000ms THEN (* automatic trigger *)
// 		trig_auto := DT_TO_UDINT(DTI) MOD (TIME_TO_UDINT(TRIG_T) / UDINT#1000) = UDINT#0;
// 	END_IF;
// END_IF;
//
// CASE step_1 OF
//
// 00:	IF ENABLE THEN
// 		aw_enable := AUTO_CLOSE >= T#5s;
// 		wd_time := SEL(X.LOAD_TIME_MAX > T#0s, T#5ms,X.LOAD_TIME_MAX);
// 		fn_last := fn; (* store current file name *)
// 		IF X.ID_MAX = USINT#0 THEN (* scan for satellite blocks only once *)
// 			X.ADD_COM := 01; (* ADD INFO *)
// 			X.STORE_TYPE := BYTE#2; (* CSV mode *)
// 		END_IF;
// 		step_1 := 10;
//
// 		(* ---------------- Debug-Message -----------------------*)
// 		(*IF _debug_enable THEN
// 			LOG_CL.NEW_MSG := 'FILE_CSV1 - Start: File [~1], [~2]';
// 			LOG_CL.PRINTF[1] := fn_last;
// 			LOG_CL.PRINTF[2] := DT_TO_STRING(DTI);
// 			LOG_MSG();
// 		END_IF;*)
// 		(* -----------------------------------------------------------------*)
//
// 	END_IF;
//
// 10:	X.UCB.D_STRING := fn_last;
// 	IF fn_last = SAVE_DATA.FN_REM THEN
// 		X.UCB.D_HEAD := WORD#16#F201; (* Filemode open + write *)
// 		X.ADD_COM := 00;
// 	ELSE
// 		X.UCB.D_HEAD := WORD#16#F301; (* Filemode create + write *)
// 		X.ADD_COM := 02; (* ADD HEADER *)
// 	END_IF;
//
// 	X.UCB.D_MODE := 1; (* store file name as string *)
// 	UCB(DATA:=X.UCB); (* enter data *)
// 	step_1 := 30;
//
// 30:	(* process LOG trigger *)
// 	trig_tmp := (TRIG_M AND NOT trig_m_last) OR trig_auto OR X.ADD_DATA_REQ;
//
// 	IF ENABLE = FALSE OR fn <> fn_last THEN (* ENABLE = 0 or new file name -> log stop *)
// 		trig_stored := trig_tmp; (* store current trigger pulse *)
// 		X.UCB.D_HEAD := WORD#16#EE00;
// 		X.UCB.D_MODE := 1;
// 		UCB(DATA:=X.UCB); (* write element *)
// 		X.ADD_COM := 00;
// 		step_1 := 00;
//
// 		(* ---------------- Debug-Message -----------------------*)
// 		(*IF _debug_enable THEN
// 			LOG_CL.NEW_MSG := 'FILE_CSV1 - Stop: [~2]';
// 			LOG_CL.PRINTF[2] := DT_TO_STRING(DTI);
// 			LOG_MSG();
// 		END_IF;*)
// 		(* -----------------------------------------------------------------*)
//
// 	ELSIF ENABLE THEN
// 		IF trig_tmp OR trig_stored THEN (* manual, automatic or external trigger *)
// 			trig_stored := FALSE;
// 			X.ADD_COM := 03; (* ADD DATA *)
// 			SAVE_DATA.TRIG_CNT := SAVE_DATA.TRIG_CNT + UDINT#1;
// 			SAVE_DATA.TRIG_CNT_TOTAL  := SAVE_DATA.TRIG_CNT_TOTAL + UDINT#1;
// 			(* ---------------- Debug-Message -----------------------*)
// 			(*IF _debug_enable THEN
// 				LOG_CL.NEW_MSG := 'FILE_CSV1 - Trig: [~2]';
// 				LOG_CL.PRINTF[2] := DT_TO_STRING(DTI);
// 				LOG_MSG();
// 			END_IF;*)
// 			(* -----------------------------------------------------------------*)
// 		ELSE
// 			X.ADD_COM := 04;	(* ADD DATA REQ *)
// 		END_IF;
// 	END_IF;
//
// END_CASE;
// X.ADD_DATA_REQ := FALSE; (* reset external request *)
//
// (* ##################################### *)
//
// CASE step_2 OF
//
// 00:	aw_ton(IN:= idx > 0 AND aw_enable, PT:= AUTO_CLOSE); (* AutoWrite Timer *)
// 	IF aw_ton.Q THEN (* time-controlled data writing *)
// 		aw_aktiv := TRUE;
// 		step_2 := 10; (* write data *)
// 		(* ---------------- Debug-Message -----------------------*)
// 		(*IF _debug_enable THEN
// 			LOG_CL.NEW_MSG := 'FILE_CSV2 - AutoWrite: [~2]';
// 			LOG_CL.PRINTF[2] := DT_TO_STRING(DTI);
// 			LOG_MSG();
// 		END_IF;*)
// 		(* -----------------------------------------------------------------*)
//
// 	ELSE
// 		wd_ton(IN:= FALSE, PT:= wd_time);
// 		wd_ton(IN:= TRUE);
// 		WHILE X.UCB.BUF_COUNT > 0 AND step_2 = 0 AND wd_ton.Q = FALSE DO
//
// 			X.UCB.D_MODE := 10;
// 			UCB(DATA:=X.UCB); (* read element, but do not remove it yet *)
// 			IF X.UCB.D_HEAD > WORD#16#F000 THEN (* F301 or F201 *)
// 				X.UCB.D_MODE := 11;
// 				UCB(DATA:=X.UCB); (* remove element *)
//
// 				FSD.MODE := WORD_TO_BYTE(SHR(SHL(X.UCB.D_HEAD,4),12)); (* 0X00 -> 000X = 3 create + write / 2 open + write *)
// 				FSD.OFFSET := UDINT#0; (* start at beginning of file *)
// 				FSD.FILENAME := X.UCB.D_STRING; (* file name *)
// 				PT.SIZE := UINT#0;
// 				SAVE_DATA.FN_REM := FSD.FILENAME; (* save current file name as retained *)
//
// 				IF FSD.MODE = BYTE#3 THEN	(* create new file -> then reset counter *)
// 					SAVE_DATA.TRIG_CNT := UDINT#0;
// 				END_IF;
//
// 				X.NEW_FILE := FSD.FILENAME;
// 				X.NEW_FILE_SIZE := UDINT#0;
// 				X.NEW_FILE_RTRIG := FALSE;
// 				step_2 := 20;
// 				(* ---------------- Debug-Message -----------------------*)
// 				(*IF _debug_enable THEN
// 					LOG_CL.NEW_MSG := 'FILE_CSV2 - Create: Mode [~1] , [~2]';
// 					LOG_CL.PRINTF[2] := DT_TO_STRING(DTI);
// 					LOG_CL.PRINTF[1] := BYTE_TO_STRING(FSD.MODE);
// 					LOG_MSG();
// 				END_IF;*)
// 				(* -----------------------------------------------------------------*)
//
// 			ELSIF X.UCB.D_HEAD = WORD#16#EE00 THEN (* LOG_STOP Command *)
// 				X.UCB.D_MODE := 11;
// 				UCB(DATA:=X.UCB); (* remove element *)
// 				log_stop := TRUE;
// 				step_2 := 10; (* write data *)
//
// 			ELSIF idx + X.UCB.D_SIZE + 2 < SIZEOF(PT.BUFFER) THEN (* buffer space available *)
// 				X.UCB.D_MODE := 11;
// 				UCB(DATA:=X.UCB); (* remove element *)
// 				(* ---------------- Debug-Message -----------------------*)
// 				(*IF _debug_enable THEN
// 					LOG_CL.NEW_MSG := 'FILE_CSV2 - BUF: TXT [~1],Pos [~2], [~3]';
// 					LOG_CL.PRINTF[1] := X.UCB.D_STRING;
// 					LOG_CL.PRINTF[2] := INT_TO_STRING(idx);
// 					LOG_CL.PRINTF[3] := DT_TO_STRING(DTI);
// 					LOG_MSG();
// 				END_IF;*)
// 				(* -----------------------------------------------------------------*)
// 				_STRING_TO_BUFFER(STR:=X.UCB.D_STRING, POS:=idx, PT:=REF(PT.BUFFER), SIZE:=SIZEOF(PT.BUFFER));
// 				idx := idx + LEN(X.UCB.D_STRING);
// 				n := n + USINT#1;
// 				IF n = X.ID_MAX THEN (* last element of a line *)
// 					n := USINT#0;
// 					PT.BUFFER[idx] := BYTE#16#0D;
// 					idx := idx + 1;
// 					PT.BUFFER[idx] := BYTE#16#0A;
// 				ELSE
// 					PT.BUFFER[idx] := SEP;
// 				END_IF;
// 				idx := idx + 1;
// 				X.NEW_FILE_SIZE := total_bytes + INT_TO_UDINT(idx);
// 			ELSE (* no space available *)
// 				step_2 := 10; (* write data *)
// 			END_IF;
// 			wd_ton();
// 		END_WHILE;
// 	END_IF;
//
// 10:	IF idx > 0 THEN (* write data *)
// 		FSD.MODE := BYTE#2; (* File_Open_Exist + File_Write *)
// 		FSD.OFFSET := UDINT#4294967294; (* 16#FFFF_FFFE -> special code: automatically append data to end of file *)
// 		PT.SIZE := INT_TO_UINT(idx); (* enter data length *)
// 		idx := 0;
// 		(* ---------------- Debug-Message -----------------------*)
// 		(*IF _debug_enable THEN
// 			LOG_CL.NEW_MSG := 'FILE_CSV2 - WriteData: Mode [~3] Size [~1] , [~2]';
// 			LOG_CL.PRINTF[1] := UINT_TO_STRING(PT.SIZE);
// 			LOG_CL.PRINTF[2] := DT_TO_STRING(DTI);
// 			LOG_CL.PRINTF[3] := BYTE_TO_STRING(FSD.MODE);
// 			LOG_MSG();
// 		END_IF;*)
// 		(* -----------------------------------------------------------------*)
// 	END_IF;
// 	step_2 := 20;
//
// 20:	IF FSD.MODE = BYTE#0 THEN
// 		total_bytes := FSD.FILE_SIZE;
// 		X.NEW_FILE_SIZE := total_bytes + INT_TO_UDINT(idx);
// 		IF log_stop OR aw_aktiv THEN
// 			aw_aktiv := FALSE;
// 			FSD.MODE := BYTE#5; (* close file *)
// 			(* ---------------- Debug-Message -----------------------*)
// 			(*IF _debug_enable THEN
// 				LOG_CL.NEW_MSG := 'FILE_CSV2 - Close: [~2]';
// 				LOG_CL.PRINTF[2] := DT_TO_STRING(DTI);
// 				LOG_MSG();
// 			END_IF;*)
// 			(* -----------------------------------------------------------------*)
// 		END_IF;
// 		step_2 := 30;
// 	END_IF;
//
// 30:	IF FSD.MODE = BYTE#0 THEN (* command finished? *)
// 		IF log_stop THEN
// 			X.NEW_FILE_RTRIG := TRUE;
// 			log_stop := FALSE;
// 			SAVE_DATA.FN_REM := ''; (* clear retained file name *)
// 		END_IF;
// 		step_2 := 00;
// 	END_IF;
//
// END_CASE;
//
// FS(FSD:=FSD,PT:=PT); (* FILE_SERVER *)
// (* error evaluation *)
// IF FSD.ERROR <> BYTE#0 THEN
// 	ERROR_C := BYTE_TO_DWORD(FSD.ERROR);
// 	ERROR_T := BYTE#1;
// ELSIF X.UCB.BUF_DATA_LOST > UDINT#0 THEN
// 	ERROR_C := DWORD#2; (* error: buffer overflow - reduce amount of data *)
// 	ERROR_T := BYTE#6; 	(* Type: Buffer *)
// ELSIF X.UCB.BUF_USED_MAX > USINT#90 THEN
// 	ERROR_C := DWORD#1; (* warning: buffer utilization > 90% *)
// 	ERROR_T := BYTE#6;	(* Type: Buffer *)
// ELSE
// 	ERROR_C := DWORD#0;
// 	ERROR_T := BYTE#0;
// END_IF;
//
// trig_m_last := TRIG_M;
// END_FUNCTION_BLOCK

// Commented out for beedance: it names a variable fn, which beedance reads as its function keyword.
// FUNCTION_BLOCK DLOG_STORE_FILE_HTML
// VAR_IN_OUT
// 	X : DLOG_DATA;
// 	SAVE_DATA : DLOG_SAVE;
// END_VAR
// VAR_INPUT
// 	ENABLE : BOOL;
// 	TRIG_M : BOOL;
// 	TRIG_T : TIME;
// 	FILENAME : STRING;
// 	DTI : DT;
// 	AUTO_CLOSE : TIME := T#15s;
// 	HTML_CAPTION : STRING;
// 	HTML_TABLE : STRING;
// 	HTML_TR_HEAD : STRING;
// 	HTML_TR_EVEN : STRING;
// 	HTML_TR_ODD : STRING;
// END_VAR
// VAR_OUTPUT
// 	ERROR_C : DWORD;
// 	ERROR_T : BYTE;
// END_VAR
// VAR
// 	FS : FILE_SERVER;
// 	FSD : FILE_SERVER_DATA;
// 	PT : NETWORK_BUFFER;
// 	UCB : UNI_CIRCULAR_BUFFER;
// 	trig_auto : BOOL;
// 	trig_stored : BOOL;
// 	trig_tmp : BOOL;
// 	trig_m_last : BOOL;
// 	dti_last : DT := DT#2070-02-06-06:28:15;
// 	fn_last : STRING;
// 	str : STRING(STRING_LENGTH);
// 	fn : STRING;
// 	step_1 : INT;
// 	step_2 : INT;
// 	idx : INT;
// 	log_state : USINT;
// 	log_stop : BOOL;
// 	n : INT;
// 	wd_ton : TON;
// 	wd_time : TIME;
// 	aw_ton : TON;
// 	aw_enable : BOOL;
// 	aw_aktiv : BOOL;
// 	total_bytes : UDINT;
// 	cur_ode : BYTE;
//
// 	(*
// 	LOG_MSG : LOG_MSG;
// 	_debug_enable : BOOL := TRUE;
// 	*)
//
// END_VAR
//
// X.DTI := DTI; (* enter date / time *)
// X.CLOCK_TRIG := DTI <> dti_last;
// dti_last := DTI;
// trig_auto := FALSE;
// IF X.CLOCK_TRIG THEN (* pulse every second *)
// 	fn := DT_TO_STRF(DTI, 0, FILENAME, 0); (* automatic file name generation *)
// 	IF TRIG_T >= T#1000ms THEN (* automatic trigger *)
// 		trig_auto := DT_TO_UDINT(DTI) MOD (TIME_TO_UDINT(TRIG_T) / UDINT#1000) = UDINT#0;
// 	END_IF;
// END_IF;
//
// CASE step_1 OF
//
// 00:	IF ENABLE THEN
// 		aw_enable := AUTO_CLOSE >= T#5s;
// 		wd_time := SEL(X.LOAD_TIME_MAX > T#0s, T#5ms,X.LOAD_TIME_MAX);
// 		fn_last := fn; (* store current file name *)
// 		IF X.ID_MAX = USINT#0 THEN (* scan for satellite blocks only once *)
// 			X.ADD_COM := 01; (* ADD INFO *)
// 			X.STORE_TYPE := BYTE#4; (* HTML mode *)
// 		END_IF;
// 		step_1 := 10;
//
// 		(* ---------------- Debug-Message -----------------------*)
// 		(*IF _debug_enable THEN
// 			LOG_CL.NEW_MSG := 'FILE_HTML1 - Start: File [~1], [~2]';
// 			LOG_CL.PRINTF[1] := fn_last;
// 			LOG_CL.PRINTF[2] := DT_TO_STRING(DTI);
// 			LOG_MSG();
// 		END_IF;*)
// 		(* -----------------------------------------------------------------*)
//
// 	END_IF;
//
// 10:	X.UCB.D_STRING := fn_last;
// 	IF fn_last = SAVE_DATA.FN_REM THEN
// 		X.UCB.D_HEAD := WORD#16#F201; (* Filemode open + write *)
// 		X.ADD_COM := 00;
// 	ELSE
// 		X.UCB.D_HEAD := WORD#16#F301; (* Filemode create + write *)
// 		X.ADD_COM := 02; (* ADD HEADER *)
// 	END_IF;
//
// 	X.UCB.D_MODE := 1; (* store file name as string *)
// 	UCB(DATA:=X.UCB); (* enter data *)
// 	step_1 := 30;
//
// 30:	(* process LOG trigger *)
// 	trig_tmp := (TRIG_M AND NOT trig_m_last) OR trig_auto OR X.ADD_DATA_REQ;
//
// 	IF ENABLE = FALSE OR fn <> fn_last THEN (* ENABLE = 0 or new file name -> log stop *)
// 		trig_stored := trig_tmp; (* store current trigger pulse *)
// 		X.UCB.D_HEAD := WORD#16#EE00;
// 		X.UCB.D_MODE := 1;
// 		UCB(DATA:=X.UCB); (* write element *)
// 		X.ADD_COM := 00;
// 		step_1 := 00;
//
// 		(* ---------------- Debug-Message -----------------------*)
// 		(*IF _debug_enable THEN
// 			LOG_CL.NEW_MSG := 'FILE_HTML1 - Stop: [~2]';
// 			LOG_CL.PRINTF[2] := DT_TO_STRING(DTI);
// 			LOG_MSG();
// 		END_IF;*)
// 		(* -----------------------------------------------------------------*)
//
// 	ELSIF ENABLE THEN
// 		IF trig_tmp OR trig_stored THEN (* manual, automatic or external trigger *)
// 			trig_stored := FALSE;
// 			X.ADD_COM := 03; (* ADD DATA *)
// 			SAVE_DATA.TRIG_CNT := SAVE_DATA.TRIG_CNT + UDINT#1;
// 			SAVE_DATA.TRIG_CNT_TOTAL  := SAVE_DATA.TRIG_CNT_TOTAL + UDINT#1;
// 			(* ---------------- Debug-Message -----------------------*)
// 			(*IF _debug_enable THEN
// 				LOG_CL.NEW_MSG := 'FILE_HTML1 - Trig: [~2]';
// 				LOG_CL.PRINTF[2] := DT_TO_STRING(DTI);
// 				LOG_MSG();
// 			END_IF;*)
// 			(* -----------------------------------------------------------------*)
// 		ELSE
// 			X.ADD_COM := 04;	(* ADD DATA REQ *)
// 		END_IF;
// 	END_IF;
//
// END_CASE;
// X.ADD_DATA_REQ := FALSE; (* reset external request *)
//
// (* ##################################### *)
//
// CASE step_2 OF
//
// 00:	aw_ton(IN:= idx > 0 AND aw_enable , PT:= AUTO_CLOSE); (* AutoWrite Timer *)
// 	IF aw_ton.Q THEN (* time-controlled data writing *)
// 		aw_aktiv := TRUE;
// 		step_2 := 10; (* write data *)
// 		(* ---------------- Debug-Message -----------------------*)
// 		(*IF _debug_enable THEN
// 			LOG_CL.NEW_MSG := 'FILE_HTML2 - AutoWrite: [~2]';
// 			LOG_CL.PRINTF[2] := DT_TO_STRING(DTI);
// 			LOG_MSG();
// 		END_IF;*)
// 		(* -----------------------------------------------------------------*)
//
// 	ELSE
// 		wd_ton(IN:= FALSE, PT:= wd_time);
// 		wd_ton(IN:= TRUE);
// 		WHILE X.UCB.BUF_COUNT > 0 AND step_2 = 0 AND wd_ton.Q = FALSE DO
//
// 			X.UCB.D_MODE := 10;
// 			UCB(DATA:=X.UCB); (* read element, but do not remove it yet *)
//
// 			IF X.UCB.D_HEAD > WORD#16#F000 THEN (* F301 or F201 *)
//
// 				str := CONCAT('<html><body><table ',HTML_TABLE);
// 		        		str := CONCAT(str,'><caption>');
// 		        		str := CONCAT(str,HTML_CAPTION);
// 		        		str := CONCAT(str,'</caption>');
//
// 				IF idx + LEN(str) < SIZEOF(PT.BUFFER) THEN (* space for element available? *)
//
// 					FSD.MODE := WORD_TO_BYTE(SHR(SHL(X.UCB.D_HEAD,4),12)); (* 0X00 -> 000X = 3 create + write / 2 open + write *)
// 					FSD.OFFSET := UDINT#0; (* start at beginning of file *)
// 					FSD.FILENAME := X.UCB.D_STRING; (* file name *)
// 					PT.SIZE := UINT#0;
// 					SAVE_DATA.FN_REM := FSD.FILENAME; (* save current file name as retained *)
//
// 					X.NEW_FILE := FSD.FILENAME;
// 					X.NEW_FILE_SIZE := UDINT#0;
// 					X.NEW_FILE_RTRIG := FALSE;
// 					step_2 := 20;
//
// 					(* write header data *)
// 					IF FSD.MODE = BYTE#3 THEN
// 						SAVE_DATA.TRIG_CNT := UDINT#0; (* create new file -> then reset counter *)
// 						SAVE_DATA.COLOR := FALSE;
// 						SAVE_DATA.HEAD := FALSE;
//
// 						_STRING_TO_BUFFER(STR:=str, POS:=idx, PT:=REF(PT.BUFFER), SIZE:=SIZEOF(PT.BUFFER));
// 						idx := idx + LEN(str);
// 						X.NEW_FILE_SIZE := total_bytes + INT_TO_UDINT(idx);
// 					END_IF;
//
// 					X.UCB.D_MODE := 11;
// 					UCB(DATA:=X.UCB); (* remove element *)
//
// 					(* ---------------- Debug-Message -----------------------*)
// 					(*IF _debug_enable THEN
// 						LOG_CL.NEW_MSG := 'FILE_HTML2 - Create: Mode [~1] , [~2]';
// 						LOG_CL.PRINTF[2] := DT_TO_STRING(DTI);
// 						LOG_CL.PRINTF[1] := BYTE_TO_STRING(FSD.MODE);
// 						LOG_MSG();
// 					END_IF;*)
// 					(* -----------------------------------------------------------------*)
// 				END_IF;
//
// 			ELSIF X.UCB.D_HEAD = WORD#16#EE00 THEN (* LOG_STOP Command *)
//
// 				str := '</table></body></html>';
//
// 				IF idx + LEN(str) < SIZEOF(PT.BUFFER) THEN (* space for element available? *)
//
// 					_STRING_TO_BUFFER(STR:=str, POS:=idx, PT:=REF(PT.BUFFER), SIZE:=SIZEOF(PT.BUFFER));
// 					idx := idx + LEN(str);
// 					log_stop := TRUE;
// 					step_2 := 10; (* write data *)
//
// 					X.UCB.D_MODE := 11;
// 					UCB(DATA:=X.UCB); (* remove element *)
// 				END_IF;
//
// 			ELSIF idx + LEN(X.UCB.D_STRING) + 120 < SIZEOF(PT.BUFFER) THEN (* space for element available? *)
//
// 				(* ---------------- Debug-Message -----------------------*)
// 				(*IF _debug_enable THEN
// 					LOG_CL.NEW_MSG := 'FILE_CSV2 - BUF: TXT [~1],Pos [~2], [~3]';
// 					LOG_CL.PRINTF[1] := X.UCB.D_STRING;
// 					LOG_CL.PRINTF[2] := INT_TO_STRING(idx);
// 					LOG_CL.PRINTF[3] := DT_TO_STRING(DTI);
// 					LOG_MSG();
// 				END_IF;*)
// 				(* -----------------------------------------------------------------*)
//
// 				IF log_state = USINT#0 THEN
// 					str := '<TR ';
// 					IF NOT SAVE_DATA.HEAD THEN
// 						str := CONCAT(str,HTML_TR_HEAD);
// 						SAVE_DATA.HEAD := TRUE;
// 					ELSIF SAVE_DATA.COLOR THEN
// 						str := CONCAT(str,HTML_TR_EVEN);
// 					ELSE
// 						str := CONCAT(str,HTML_TR_ODD);
// 					END_IF;
// 					str := CONCAT(str,'><TD>');
// 				ELSE
// 					str := '<TD>';
// 				END_IF;
//
// 				_STRING_TO_BUFFER(STR:=str, POS:=idx, PT:=REF(PT.BUFFER), SIZE:=SIZEOF(PT.BUFFER));
// 				idx := idx + LEN(str);
// 				log_state := log_state + USINT#1;
//
// 				_STRING_TO_BUFFER(STR:=X.UCB.D_STRING, POS:=idx, PT:=REF(PT.BUFFER), SIZE:=SIZEOF(PT.BUFFER));
// 				idx := idx + LEN(X.UCB.D_STRING);
// 				n := n + USINT#1;
// 				IF n >= X.ID_MAX THEN
// 					n := USINT#0;
// 					str := '</TD></TR>';
// 					SAVE_DATA.COLOR := NOT SAVE_DATA.COLOR;
// 					log_state := USINT#0;
// 				ELSE
// 					str := '</TD>';
// 				END_IF;
// 				_STRING_TO_BUFFER(STR:=str, POS:=idx, PT:=REF(PT.BUFFER), SIZE:=SIZEOF(PT.BUFFER));
// 				idx := idx + LEN(str);
// 				X.NEW_FILE_SIZE := total_bytes + INT_TO_UDINT(idx);
//
// 				X.UCB.D_MODE := 11;
// 				UCB(DATA:=X.UCB); (* remove element *)
//
// 			ELSE (* no space available *)
// 				step_2 := 10; (* write data *)
//
// 			END_IF;
// 			wd_ton();
// 		END_WHILE;
// 	END_IF;
//
// 10:	IF idx > 0 THEN (* write data *)
// 		FSD.MODE := BYTE#2; (* File_Open_Exist + File_Write *)
// 		FSD.OFFSET := UDINT#4294967294; (* 16#FFFF_FFFE -> special code: automatically append data to end of file *)
// 		PT.SIZE := INT_TO_UINT(idx); (* enter data length *)
// 		idx := 0;
// 		(* ---------------- Debug-Message -----------------------*)
// 		(*IF _debug_enable THEN
// 			LOG_CL.NEW_MSG := 'FILE_HTML2 - WriteData: Mode [~3] Size [~1] , [~2]';
// 			LOG_CL.PRINTF[1] := UINT_TO_STRING(PT.SIZE);
// 			LOG_CL.PRINTF[2] := DT_TO_STRING(DTI);
// 			LOG_CL.PRINTF[3] := BYTE_TO_STRING(FSD.MODE);
// 			LOG_MSG();
// 		END_IF;*)
// 		(* -----------------------------------------------------------------*)
// 	END_IF;
// 	step_2 := 20;
//
// 20:	IF FSD.MODE = BYTE#0 THEN
// 		total_bytes := FSD.FILE_SIZE;
// 		X.NEW_FILE_SIZE := total_bytes + INT_TO_UDINT(idx);
// 		IF log_stop OR aw_aktiv THEN
// 			aw_aktiv := FALSE;
// 			FSD.MODE := BYTE#5; (* close file *)
// 			(* ---------------- Debug-Message -----------------------*)
// 			(*IF _debug_enable THEN
// 				LOG_CL.NEW_MSG := 'FILE_HTML2 - Close: [~2]';
// 				LOG_CL.PRINTF[2] := DT_TO_STRING(DTI);
// 				LOG_MSG();
// 			END_IF;*)
// 			(* -----------------------------------------------------------------*)
// 		END_IF;
// 		step_2 := 30;
// 	END_IF;
//
// 30:	IF FSD.MODE = BYTE#0 THEN (* file close finished *)
// 		IF log_stop THEN
// 			X.NEW_FILE_RTRIG := TRUE;
// 			log_stop := FALSE;
// 			SAVE_DATA.FN_REM := ''; (* clear retained file name *)
// 		END_IF;
// 		step_2 := 00;
// 	END_IF;
//
// END_CASE;
//
// FS(FSD:=FSD,PT:=PT); (* FILE_SERVER *)
//
// (* error evaluation *)
// IF FSD.ERROR <> BYTE#0 THEN
// 	ERROR_C := BYTE_TO_DWORD(FSD.ERROR);
// 	ERROR_T := BYTE#1;
// ELSIF X.UCB.BUF_DATA_LOST > UDINT#0 THEN
// 	ERROR_C := DWORD#2; (* error: buffer overflow - reduce amount of data *)
// 	ERROR_T := BYTE#6; 	(* Type: Buffer *)
// ELSIF X.UCB.BUF_USED_MAX > USINT#90 THEN
// 	ERROR_C := DWORD#1; (* warning: buffer utilization > 90% *)
// 	ERROR_T := BYTE#6;	(* Type: Buffer *)
// ELSE
// 	ERROR_C := DWORD#0;
// 	ERROR_T := BYTE#0;
// END_IF;
//
// trig_m_last := TRIG_M;
// END_FUNCTION_BLOCK

// Commented out for beedance: it names a variable fn, which beedance reads as its function keyword.
// FUNCTION_BLOCK DLOG_STORE_FILE_XML
// VAR_IN_OUT
// 	X : DLOG_DATA;
// 	SAVE_DATA : DLOG_SAVE;
// END_VAR
// VAR_INPUT
// 	ENABLE : BOOL;
// 	TRIG_M : BOOL;
// 	TRIG_T : TIME;
// 	FILENAME : STRING;
// 	DTI : DT;
// 	AUTO_CLOSE : TIME := T#15s;
// END_VAR
// VAR_OUTPUT
// 	ERROR_C : DWORD;
// 	ERROR_T : BYTE;
// END_VAR
// VAR
// 	FS : FILE_SERVER;
// 	FSD : FILE_SERVER_DATA;
// 	PT : NETWORK_BUFFER;
// 	UCB : UNI_CIRCULAR_BUFFER;
// 	trig_auto : BOOL;
// 	trig_stored : BOOL;
// 	trig_tmp : BOOL;
// 	trig_m_last : BOOL;
// 	dti_last : DT := DT#2070-02-06-06:28:15;
// 	fn_last : STRING;
// 	fn : STRING;
// 	str : STRING(STRING_LENGTH);
// 	step_1 : INT;
// 	step_2 : INT;
// 	idx : INT;
// 	log_state : USINT;
// 	log_stop : BOOL;
// 	n : INT;
// 	wd_ton : TON;
// 	wd_time : TIME;
// 	aw_ton : TON;
// 	aw_enable : BOOL;
// 	aw_aktiv : BOOL;
// 	total_bytes : UDINT;
//
// 	(*
// 	LOG_MSG : LOG_MSG;
// 	_debug_enable : BOOL := TRUE;
// 	*)
// END_VAR
//
// X.DTI := DTI; (* enter date / time *)
// X.CLOCK_TRIG := DTI <> dti_last;
// dti_last := DTI;
// trig_auto := FALSE;
// IF X.CLOCK_TRIG THEN (* pulse every second *)
// 	fn := DT_TO_STRF(DTI, 0, FILENAME, 0); (* automatic file name generation *)
// 	IF TRIG_T >= T#1000ms THEN (* automatic trigger *)
// 		trig_auto := DT_TO_UDINT(DTI) MOD (TIME_TO_UDINT(TRIG_T) / UDINT#1000) = UDINT#0;
// 	END_IF;
// END_IF;
//
// CASE step_1 OF
//
// 00:	IF ENABLE THEN
// 		aw_enable := AUTO_CLOSE >= T#5s;
// 		wd_time := SEL(X.LOAD_TIME_MAX > T#0s, T#5ms,X.LOAD_TIME_MAX);
// 		fn_last := fn; (* store current file name *)
// 		IF X.ID_MAX = USINT#0 THEN (* scan for satellite blocks only once *)
// 			X.ADD_COM := 01; (* ADD INFO *)
// 			X.STORE_TYPE := BYTE#3; (* XML mode *)
// 		END_IF;
// 		step_1 := 10;
//
// 		(* ---------------- Debug-Message -----------------------*)
// 		(*IF _debug_enable THEN
// 			LOG_CL.NEW_MSG := 'FILE_XML1 - Start: File [~1], [~2]';
// 			LOG_CL.PRINTF[1] := fn_last;
// 			LOG_CL.PRINTF[2] := DT_TO_STRING(DTI);
// 			LOG_MSG();
// 		END_IF;*)
// 		(* -----------------------------------------------------------------*)
//
// 	END_IF;
//
// 10:	X.UCB.D_STRING := fn_last;
// 	IF fn_last = SAVE_DATA.FN_REM THEN
// 		X.UCB.D_HEAD := WORD#16#F201; (* Filemode open + write *)
// 		X.ADD_COM := 00;
// 	ELSE
// 		X.UCB.D_HEAD := WORD#16#F301; (* Filemode create + write *)
// 		X.ADD_COM := 02; (* ADD HEADER *)
// 	END_IF;
//
// 	X.UCB.D_MODE := 1; (* store file name as string *)
// 	UCB(DATA:=X.UCB); (* enter data *)
// 	step_1 := 30;
//
// 30:	(* process LOG trigger *)
// 	trig_tmp := (TRIG_M AND NOT trig_m_last) OR trig_auto OR X.ADD_DATA_REQ;
//
// 	IF ENABLE = FALSE OR fn <> fn_last THEN (* ENABLE = 0 or new file name -> log stop *)
// 		trig_stored := trig_tmp; (* store current trigger pulse *)
// 		X.UCB.D_HEAD := WORD#16#EE00;
// 		X.UCB.D_MODE := 1;
// 		UCB(DATA:=X.UCB); (* write element *)
// 		X.ADD_COM := 00;
// 		step_1 := 00;
//
// 		(* ---------------- Debug-Message -----------------------*)
// 		(*IF _debug_enable THEN
// 			LOG_CL.NEW_MSG := 'FILE_XML1 - Stop: [~2]';
// 			LOG_CL.PRINTF[2] := DT_TO_STRING(DTI);
// 			LOG_MSG();
// 		END_IF;*)
// 		(* -----------------------------------------------------------------*)
//
// 	ELSIF ENABLE THEN
// 		IF trig_tmp OR trig_stored THEN (* manual, automatic or external trigger *)
// 			trig_stored := FALSE;
// 			X.ADD_COM := 03; (* ADD DATA *)
// 			SAVE_DATA.TRIG_CNT := SAVE_DATA.TRIG_CNT + UDINT#1;
// 			SAVE_DATA.TRIG_CNT_TOTAL  := SAVE_DATA.TRIG_CNT_TOTAL + UDINT#1;
// 			(* ---------------- Debug-Message -----------------------*)
// 			(*IF _debug_enable THEN
// 				LOG_CL.NEW_MSG := 'FILE_XML1 - Trig: [~2]';
// 				LOG_CL.PRINTF[2] := DT_TO_STRING(DTI);
// 				LOG_MSG();
// 			END_IF;*)
// 			(* -----------------------------------------------------------------*)
// 		ELSE
// 			X.ADD_COM := 04;	(* ADD DATA REQ *)
// 		END_IF;
// 	END_IF;
//
// END_CASE;
// X.ADD_DATA_REQ := FALSE; (* reset external request *)
//
// (* ##################################### *)
//
// CASE step_2 OF
//
// 00:	aw_ton(IN:= idx > 0 AND aw_enable , PT:= AUTO_CLOSE); (* AutoWrite Timer *)
// 	IF aw_ton.Q THEN (* time-controlled data writing *)
// 		aw_aktiv := TRUE;
// 		step_2 := 10; (* write data *)
// 		(* ---------------- Debug-Message -----------------------*)
// 		(*IF _debug_enable THEN
// 			LOG_CL.NEW_MSG := 'FILE_XML2 - AutoWrite: [~2]';
// 			LOG_CL.PRINTF[2] := DT_TO_STRING(DTI);
// 			LOG_MSG();
// 		END_IF;*)
// 		(* -----------------------------------------------------------------*)
//
// 	ELSE
// 		wd_ton(IN:= FALSE, PT:= wd_time);
// 		wd_ton(IN:= TRUE);
// 		WHILE X.UCB.BUF_COUNT > 0 AND step_2 = 0 AND wd_ton.Q = FALSE DO
//
// 			X.UCB.D_MODE := 10;
// 			UCB(DATA:=X.UCB); (* read element, but do not remove it yet *)
//
// 			IF X.UCB.D_HEAD > WORD#16#F000 THEN (* F301 or F201 *)
//
// 				str := '<?xml version="1.0" encoding="UTF-8"?><table>';
//
// 				IF idx + LEN(str) < SIZEOF(PT.BUFFER) THEN (* space for element available? *)
//
// 					FSD.MODE := WORD_TO_BYTE(SHR(SHL(X.UCB.D_HEAD,4),12)); (* 0X00 -> 000X = 3 create + write / 2 open + write *)
// 					FSD.OFFSET := UDINT#0; (* start at beginning of file *)
// 					FSD.FILENAME := X.UCB.D_STRING; (* file name *)
// 					PT.SIZE := UINT#0;
// 					SAVE_DATA.FN_REM := FSD.FILENAME; (* save current file name as retained *)
//
// 					X.NEW_FILE := FSD.FILENAME;
// 					X.NEW_FILE_SIZE := UDINT#0;
// 					X.NEW_FILE_RTRIG := FALSE;
// 					step_2 := 20;
//
// 					(* write header data *)
// 					IF FSD.MODE = BYTE#3 THEN
// 						SAVE_DATA.TRIG_CNT := UDINT#0; (* create new file -> then reset counter *)
//
// 						_STRING_TO_BUFFER(STR:=str, POS:=idx, PT:=REF(PT.BUFFER), SIZE:=SIZEOF(PT.BUFFER));
// 						idx := idx + LEN(str);
// 						X.NEW_FILE_SIZE := total_bytes + INT_TO_UDINT(idx);
// 					END_IF;
//
// 					X.UCB.D_MODE := 11;
// 					UCB(DATA:=X.UCB); (* remove element *)
//
// 					(* ---------------- Debug-Message -----------------------*)
// 					(*IF _debug_enable THEN
// 						LOG_CL.NEW_MSG := 'FILE_XML2 - Create: Mode [~1] , [~2]';
// 						LOG_CL.PRINTF[2] := DT_TO_STRING(DTI);
// 						LOG_CL.PRINTF[1] := BYTE_TO_STRING(FSD.MODE);
// 						LOG_MSG();
// 					END_IF;*)
// 					(* -----------------------------------------------------------------*)
// 				END_IF;
//
// 			ELSIF X.UCB.D_HEAD = WORD#16#EE00 THEN (* LOG_STOP Command *)
//
// 				str := '</table>';
//
// 				IF idx + LEN(str) < SIZEOF(PT.BUFFER) THEN (* space for element available? *)
//
// 					_STRING_TO_BUFFER(STR:=str, POS:=idx, PT:=REF(PT.BUFFER), SIZE:=SIZEOF(PT.BUFFER));
// 					idx := idx + LEN(str);
// 					log_stop := TRUE;
// 					step_2 := 10; (* write data *)
//
// 					X.UCB.D_MODE := 11;
// 					UCB(DATA:=X.UCB); (* remove element *)
//
// 				END_IF;
//
// 			ELSIF idx + LEN(X.UCB.D_STRING) + 120 < SIZEOF(PT.BUFFER) THEN (* space for element available? *)
//
// 				(* ---------------- Debug-Message -----------------------*)
// 				(*IF _debug_enable THEN
// 					LOG_CL.NEW_MSG := 'FILE_XML2 - BUF: TXT [~1],Pos [~2], [~3]';
// 					LOG_CL.PRINTF[1] := X.UCB.D_STRING;
// 					LOG_CL.PRINTF[2] := INT_TO_STRING(idx);
// 					LOG_CL.PRINTF[3] := DT_TO_STRING(DTI);
// 					LOG_MSG();
// 				END_IF;*)
// 				(* -----------------------------------------------------------------*)
//
// 				IF log_state = USINT#0 THEN
// 					str := '<row><entry>';
// 				ELSE
// 					str := '<entry>';
// 				END_IF;
//
// 				_STRING_TO_BUFFER(STR:=str, POS:=idx, PT:=REF(PT.BUFFER), SIZE:=SIZEOF(PT.BUFFER));
// 				idx := idx + LEN(str);
// 				log_state := log_state + USINT#1;
//
// 				_STRING_TO_BUFFER(STR:=X.UCB.D_STRING, POS:=idx, PT:=REF(PT.BUFFER), SIZE:=SIZEOF(PT.BUFFER));
// 				idx := idx + LEN(X.UCB.D_STRING);
//
// 				n := n + USINT#1;
// 				IF n >= X.ID_MAX THEN
// 					n := USINT#0;
// 					str := '</entry></row>';
// 					log_state := USINT#0;
// 				ELSE
// 					str := '</entry>';
// 				END_IF;
// 				_STRING_TO_BUFFER(STR:=str, POS:=idx, PT:=REF(PT.BUFFER), SIZE:=SIZEOF(PT.BUFFER));
// 				idx := idx + LEN(str);
// 				X.NEW_FILE_SIZE := total_bytes + INT_TO_UDINT(idx);
//
// 				X.UCB.D_MODE := 11;
// 				UCB(DATA:=X.UCB); (* remove element *)
//
// 			ELSE (* no space available *)
// 				step_2 := 10; (* write data *)
// 			END_IF;
// 			wd_ton();
// 		END_WHILE;
// 	END_IF;
//
// 10:	IF idx > 0 THEN (* write data *)
// 		FSD.MODE := BYTE#2; (* File_Open_Exist + File_Write *)
// 		FSD.OFFSET := UDINT#4294967294; (* 16#FFFF_FFFE -> special code: automatically append data to end of file *)
// 		PT.SIZE := INT_TO_UINT(idx); (* enter data length *)
// 		idx := 0;
// 		(* ---------------- Debug-Message -----------------------*)
// 		(*IF _debug_enable THEN
// 			LOG_CL.NEW_MSG := 'FILE_XML2 - WriteData: Mode [~3] Size [~1] , [~2]';
// 			LOG_CL.PRINTF[1] := UINT_TO_STRING(PT.SIZE);
// 			LOG_CL.PRINTF[2] := DT_TO_STRING(DTI);
// 			LOG_CL.PRINTF[3] := BYTE_TO_STRING(FSD.MODE);
// 			LOG_MSG();
// 		END_IF;*)
// 		(* -----------------------------------------------------------------*)
// 	END_IF;
// 	step_2 := 20;
//
// 20:	IF FSD.MODE = BYTE#0 THEN
// 		total_bytes := FSD.FILE_SIZE;
// 		X.NEW_FILE_SIZE := total_bytes + INT_TO_UDINT(idx);
// 		IF log_stop OR aw_aktiv THEN
// 			aw_aktiv := FALSE;
// 			FSD.MODE := BYTE#5; (* close file *)
// 			(* ---------------- Debug-Message -----------------------*)
// 			(*IF _debug_enable THEN
// 				LOG_CL.NEW_MSG := 'FILE_XML2 - Close: [~2]';
// 				LOG_CL.PRINTF[2] := DT_TO_STRING(DTI);
// 				LOG_MSG();
// 			END_IF;*)
// 			(* -----------------------------------------------------------------*)
// 		END_IF;
// 		step_2 := 30;
// 	END_IF;
//
// 30:	IF FSD.MODE = BYTE#0 THEN (* file close finished *)
// 		IF log_stop THEN
// 			X.NEW_FILE_RTRIG := TRUE;
// 			log_stop := FALSE;
// 			SAVE_DATA.FN_REM := ''; (* clear retained file name *)
// 		END_IF;
// 		step_2 := 00;
// 	END_IF;
//
// END_CASE;
//
// FS(FSD:=FSD,PT:=PT); (* FILE_SERVER *)
//
// (* error evaluation *)
// IF FSD.ERROR <> BYTE#0 THEN
// 	ERROR_C := BYTE_TO_DWORD(FSD.ERROR);
// 	ERROR_T := BYTE#1;
// ELSIF X.UCB.BUF_DATA_LOST > UDINT#0 THEN
// 	ERROR_C := DWORD#2; (* error: buffer overflow - reduce amount of data *)
// 	ERROR_T := BYTE#6; 	(* Type: Buffer *)
// ELSIF X.UCB.BUF_USED_MAX > USINT#90 THEN
// 	ERROR_C := DWORD#1; (* warning: buffer utilization > 90% *)
// 	ERROR_T := BYTE#6;	(* Type: Buffer *)
// ELSE
// 	ERROR_C := DWORD#0;
// 	ERROR_T := BYTE#0;
// END_IF;
//
// trig_m_last := TRIG_M;
// END_FUNCTION_BLOCK

// Commented out for beedance: it uses UNI_CIRCULAR_BUFFER, which is commented out.
// FUNCTION_BLOCK DLOG_STORE_MYSQL
// VAR_IN_OUT
// 	SQL_INFO : MYSQL_INFO;
// 	X : DLOG_DATA;
// END_VAR
// VAR_INPUT
// 	ENABLE : BOOL;
// 	TRIG_M : BOOL;
// 	TRIG_T : TIME;
// 	DTI : DT;
// 	URL : STRING(STRING_LENGTH);
// 	DB_NAME : STRING(64);
// 	TB_NAME : STRING(64);
// 	AUTO_DELETE : UDINT;
// 	TIMEOUT : TIME;
// 	DNS_IP4 : DWORD;
// END_VAR
// VAR_OUTPUT
// 	ERROR_C : DWORD;
// 	ERROR_T : BYTE;
// END_VAR
// VAR
// 	UCB : UNI_CIRCULAR_BUFFER;
// 	MYSQL_CONTROL: MYSQL_CONTROL;
// 	trig_auto : BOOL;
// 	trig_tmp : BOOL;
// 	trig_m_last : BOOL;
// 	dti_last : DT := DT#2070-02-06-06:28:15;
// 	enable_last : BOOL;
// 	step : INT;
// 	idx : INT;
// 	n : USINT;
// 	snd_text : STRING(STRING_LENGTH);
// 	snd_size : INT;
// 	sql_command : BYTE;
// 	next_step : INT;
// 	i1 : INT;
// 	i2 : INT;
// 	y: MYSQL_COM;
// 	del_dt : UDINT;
// 	del_start : BOOL;
// 	run : BOOL;
//
// 	(*
// 	LOG_MSG : LOG_MSG;
// 	_debug_enable : BOOL := TRUE;
// 	*)
// END_VAR
//
// X.DTI := DTI; (* enter date / time *)
// X.CLOCK_TRIG := DTI <> dti_last;
// dti_last := DTI;
// trig_auto := FALSE;
// IF X.CLOCK_TRIG THEN (* pulse every second *)
// 	del_start := DT_TO_UDINT(DTI) - del_dt > AUTO_DELETE AND AUTO_DELETE > UDINT#0;
// 	IF TRIG_T >= T#1000ms THEN (* automatic trigger *)
// 		trig_auto := DT_TO_UDINT(DTI) MOD (TIME_TO_UDINT(TRIG_T) / UDINT#1000) = UDINT#0;
// 	END_IF;
// END_IF;
// X.ADD_COM := 00;
//
// CASE step OF
//
// 00:	IF ENABLE AND enable_last = FALSE THEN
// 		y.SQL_URL := URL;
// 		y.TIMEOUT := TIMEOUT;
// 		y.DNS_IP4 := DNS_IP4;
// 		y.SQL_CON := TRUE;
//
// 		X.UCB.D_MODE := 99; (* buffer reset - delete everything *)
// 		UCB(DATA:=X.UCB);
//
// 		IF X.ID_MAX = USINT#0 THEN (* scan for satellite blocks only once *)
// 			X.ADD_COM := 01; (* ADD INFO *)
// 			X.STORE_TYPE := BYTE#5; (* MySQL mode *)
// 		END_IF;
//
// 		step := 05;
// 	END_IF;
//
// 05:	X.ADD_COM := 02; (* ADD HEADER *)
// 	step := 10;
//
// 10:	IF SQL_INFO.SQL_CONNECTED THEN
// 		sql_command := BYTE#3; (* CREATE DATABASE IF NOT EXISTS `db_name` *)
// 		snd_text :=  CONCAT('CREATE DATABASE IF NOT EXISTS `' ,DB_NAME);
// 		snd_text :=  CONCAT(snd_text, '`');
// 		next_step := 20;
// 	END_IF;
//
// 20:	sql_command := BYTE#2; (* 0x02 COM_INIT_DB mysql_select_db *)
// 	snd_text := DB_NAME;
// 	next_step := 30;
//
// 30:	(* CREATE TABLE IF NOT EXISTS tb_name (Timestamp TIMESTAMP NULL DEFAULT CURRENT_TIMESTAMP, n1,n2) *)
// 	sql_command := BYTE#0;
// 	idx := 5;
// 	n := USINT#0;
// 	WHILE sql_command = BYTE#0 DO
// 		IF n = USINT#0 THEN
// 			snd_text := CONCAT('CREATE TABLE IF NOT EXISTS `', TB_NAME);
// 			snd_text := CONCAT(snd_text,'` (`ID` BIGINT NOT NULL AUTO_INCREMENT PRIMARY KEY ,');
// 			snd_text := CONCAT(snd_text,' store_timestamp TIMESTAMP NULL DEFAULT CURRENT_TIMESTAMP');
// 		ELSIF n <= X.ID_MAX THEN
// 			X.UCB.D_MODE := 12; (* read and delete element *)
// 			UCB(DATA:=X.UCB);
// 			snd_text := CONCAT(', `',X.UCB.D_STRING);
// 			CASE WORD_TO_INT(SHR(X.UCB.D_HEAD,8)) OF
// 			02:	snd_text := CONCAT(snd_text, '` FLOAT'); (* REAL *)
// 			06:	snd_text := CONCAT(snd_text, '` BOOL'); (* BOOL *)
// 			08:	snd_text := CONCAT(snd_text, '` INT'); (* DINT *)
// 			13:	snd_text := CONCAT(snd_text, '` DATETIME'); (* DT *)
// 			ELSE
// 				snd_text := CONCAT(snd_text, '` VARCHAR(80)'); (* STRING(80) *)
// 			END_CASE;
// 		ELSE
// 			snd_text := ')';
// 			sql_command := BYTE#3;
// 			snd_size := idx + LEN(snd_text);
// 			next_step := 40;
// 		END_IF;
// 		_STRING_TO_BUFFER(str:=snd_text,pos:=idx,pt:=REF(y.S_BUF.BUFFER),size:=SIZEOF(y.S_BUF.BUFFER)); (* copy string into buffer *)
// 		idx := idx + LEN(snd_text);
// 		n := n + USINT#1;
//
// 		(*####################  DEBUG-MESSAGE  ###################################*)
// 		(*IF _debug_enable THEN
// 			LOG_CL.NEW_MSG := 'dlog_mysql: create >~1<';
// 			LOG_CL.PRINTF[1] := snd_text;
// 			LOG_MSG();
// 		END_IF;*)
// 		(*########################################################################*)
// 	END_WHILE;
//
// 40:	IF del_start THEN
// 		del_start := FALSE;
// 		sql_command := BYTE#3; (* DELETE FROM `tb_name` WHERE TIMESTAMPDIFF(SECOND, Timestamp, NOW()) > xxx *)
// 		snd_text := CONCAT('DELETE FROM `', TB_NAME);
// 		snd_text := CONCAT(snd_text, '` WHERE TIMESTAMPDIFF(SECOND, store_timestamp, NOW()) > ');
// 		snd_text := CONCAT(snd_text, UDINT_TO_STRING(AUTO_DELETE));
// 		next_step := 40;
// 		del_dt := DT_TO_UDINT(DTI);
// 		(*####################  DEBUG-MESSAGE  ###################################*)
// 		(*IF _debug_enable THEN
// 			LOG_CL.NEW_MSG := 'dlog_mysql: # delete time:~1 >~2<';
// 			LOG_CL.PRINTF[1] := UDINT_TO_STRING(AUTO_DELETE);
// 			LOG_CL.PRINTF[2] := snd_text;
// 			LOG_MSG();
// 		END_IF;*)
// 		(*########################################################################*)
//
//          (* INSERT INTO `tb_name` VALUES (CURRENT_TIMESTAMP,  "n1","n2") *)
// 	ELSIF X.UCB.BUF_COUNT >= USINT_TO_INT(X.ID_MAX) AND step > 0 THEN (* new data row(s) available *)
// 		idx := 5;
// 		n := USINT#0;
// 		sql_command := BYTE#0;
// 		WHILE sql_command = BYTE#0 DO
// 			IF n = USINT#0 THEN
// 				snd_text := CONCAT('INSERT INTO `', TB_NAME);
// 				snd_text := CONCAT(snd_text,'` VALUES (NULL, CURRENT_TIMESTAMP');
// 			ELSIF n <= X.ID_MAX THEN
// 				X.UCB.D_MODE := 12; (* read and delete element *)
// 				UCB(DATA:=X.UCB);
// 				snd_text := CONCAT(', "',X.UCB.D_STRING);
// 				snd_text := CONCAT(snd_text, '"');
// 			ELSE
// 				snd_text := ')';
// 				sql_command := BYTE#3;
// 				snd_size := idx + LEN(snd_text);
// 				next_step := 40;
// 			END_IF;
// 			_STRING_TO_BUFFER(str:=snd_text,pos:=idx,pt:=REF(y.S_BUF.BUFFER),size:=SIZEOF(y.S_BUF.BUFFER)); (* copy string into buffer *)
// 			idx := idx + LEN(snd_text);
// 			n := n + USINT#1;
//
// 			(*####################  DEBUG-MESSAGE  ###################################*)
// 			(*IF _debug_enable THEN
// 				LOG_CL.NEW_MSG := 'dlog_mysql: insert >~1<';
// 				LOG_CL.PRINTF[1] := snd_text;
// 				LOG_MSG();
// 			END_IF;*)
// 			(*########################################################################*)
// 		END_WHILE;
// 	END_IF;
//
// 	IF ENABLE THEN 	(* process LOG trigger *)
// 		trig_tmp := (TRIG_M AND NOT trig_m_last) OR trig_auto OR X.ADD_DATA_REQ;
//
// 		IF trig_tmp THEN (* manual, automatic or external trigger *)
// 			X.ADD_COM := 03; (* ADD DATA *)
// 			(* ---------------- Debug-Message -----------------------*)
// 			(*IF _debug_enable THEN
// 				LOG_CL.NEW_MSG := 'dlog_mysql: Trigger: DATE [~2]';
// 				LOG_CL.PRINTF[2] := DT_TO_STRING(DTI);
// 				LOG_MSG();
// 			END_IF;*)
// 			(* -----------------------------------------------------------------*)
// 		ELSE
// 			X.ADD_COM := 04;	(* ADD DATA REQ *)
// 		END_IF;
// 	ELSE
// 		y.SQL_CON := FALSE; (* close MySQL connection *)
// 		step := 0;
// 	END_IF;
// 	X.ADD_DATA_REQ := FALSE;
//
// (* ~~~~~~~~~~~~~~~~~~~~~~ *)
//
// 199:IF y.SQL_RCV_STATE = BYTE#1 THEN (* OK *)
// 		step := next_step;
// 	ELSIF y.SQL_RCV_STATE = BYTE#2 THEN  (* ERROR *)
// 		step := 0;
// 	END_IF;
//
// END_CASE;
//
// (* ########################## *)
// (* execute SQL command *)
// IF sql_command > BYTE#0 THEN
//
// 	IF snd_size > 0 THEN
// 		y.S_BUF.SIZE := INT_TO_UINT(snd_size);
// 		snd_size := 0;
// 	ELSE
// 		_STRING_TO_BUFFER(str:=snd_text,pos:=5,pt:=REF(y.S_BUF.BUFFER),size:=SIZEOF(y.S_BUF.BUFFER)); (* copy string into buffer *)
// 		y.S_BUF.SIZE := INT_TO_UINT(5 + LEN(snd_text));
// 		snd_text := '';
// 	END_IF;
//
// 	IF y.S_BUF.SIZE > SIZEOF(y.S_BUF.BUFFER) THEN (* buffer overflow detected -> abort *)
// 		y.S_BUF.SIZE := 0;
// 		sql_command := BYTE#0;
// 		y.SQL_CON := FALSE; (* close MySQL connection *)
// 		step := 999; (* dummy step *)
// 	ELSE
//
// 		i2 := UINT_TO_INT(y.S_BUF.SIZE) - 1; (* replace all " characters with ' *)
// 		FOR i1 := 5 TO i2 DO
// 			IF y.S_BUF.BUFFER[i1] = BYTE#34 THEN
// 				y.S_BUF.BUFFER[i1] := BYTE#39;
// 			END_IF;
// 		END_FOR;
//
// 		y.S_BUF.BUFFER[4] := sql_command;
// 		y.SQL_PACKET_NO := BYTE#255;
// 		sql_command := BYTE#0;
// 		step := 199;
// 	END_IF;
// END_IF;
//
// (* ########################## *)
//
// MYSQL_CONTROL(COM:= y, INFO:=SQL_INFO);
//
// (* error evaluation *)
// IF step = 999 THEN	(* buffer overflow *)
// 	ERROR_C := DWORD#3; (* network buffer overflow *)
// 	ERROR_T := BYTE#6; 	(* Type: Buffer *)
// ELSIF y.ERROR_T > BYTE#0 THEN	(* SQL Error *)
// 	ERROR_C := y.ERROR_C;
// 	ERROR_T := y.ERROR_T;
// 	step := 0;
// ELSIF X.UCB.BUF_DATA_LOST > UDINT#0 THEN
// 	ERROR_C := DWORD#2; (* error: buffer overflow - reduce amount of data *)
// 	ERROR_T := BYTE#6; 	(* Type: Buffer *)
// ELSIF X.UCB.BUF_USED_MAX > USINT#90 THEN
// 	ERROR_C := DWORD#1; (* warning: buffer utilization > 90% *)
// 	ERROR_T := BYTE#6;	(* Type: Buffer *)
// ELSE
// 	ERROR_C := DWORD#0;
// 	ERROR_T := BYTE#0;
// END_IF;
//
// (* ########################## *)
//
// trig_m_last := TRIG_M;
// enable_last := ENABLE;
// run := step > 0;
// END_FUNCTION_BLOCK

// Commented out for beedance: it uses UNI_CIRCULAR_BUFFER, which is commented out.
// FUNCTION_BLOCK DLOG_STORE_RRD
// VAR_IN_OUT
// 	X : DLOG_DATA;
// END_VAR
// VAR_INPUT
// 	ENABLE : BOOL;
// 	TRIG_M : BOOL;
// 	TRIG_T : TIME;
// 	URL : STRING(STRING_LENGTH);
// 	DTI : DT;
// 	SEP : BYTE;
// 	DNS_IP4 : DWORD;
// 	TIMEOUT : TIME;
// END_VAR
// VAR_OUTPUT
// 	ERROR_C : DWORD;
// 	ERROR_T : BYTE;
// END_VAR
// VAR
// 	UCB : UNI_CIRCULAR_BUFFER;
// 	IP_C : IP_C; (* IP_Control management structure *)
// 	S_BUF : NETWORK_BUFFER;
// 	R_BUF : NETWORK_BUFFER;
// 	URL_DATA : url;
// 	DNS_CLIENT : DNS_CLIENT;
// 	HTTP_GET : HTTP_GET;
// 	IPC : IP_CONTROL;
//
// 	trig_auto : BOOL;
// 	trig_stored : BOOL;
// 	trig_tmp : BOOL;
// 	trig_m_last : BOOL;
// 	dti_last : DT := DT#2070-02-06-06:28:15;
// 	step_1 : INT;
// 	step_2 : INT;
// 	sep_char : STRING(1);
// 	url_query : STRING(STRING_LENGTH);
// 	n : INT;
//
// 	(*
// 	LOG_MSG : LOG_MSG;
// 	_debug_enable : BOOL := TRUE;
// 	*)
// END_VAR
//
// X.DTI := DTI; (* enter date / time *)
// X.CLOCK_TRIG := DTI <> dti_last;
// dti_last := DTI;
// trig_auto := FALSE;
// IF X.CLOCK_TRIG THEN (* pulse every second *)
// 	IF TRIG_T >= T#1000ms THEN (* automatic trigger *)
// 		trig_auto := DT_TO_UDINT(DTI) MOD (TIME_TO_UDINT(TRIG_T) / UDINT#1000) = UDINT#0;
// 	END_IF;
// END_IF;
//
// CASE step_1 OF
//
// 00:	IF ENABLE THEN
// 		IF X.ID_MAX = USINT#0 THEN (* scan for satellite blocks only once *)
// 			X.ADD_COM := 01; (* ADD INFO *)
// 			X.STORE_TYPE := BYTE#1; (* RRD mode *)
// 		END_IF;
//
// 		ERROR_T := BYTE#0;
// 		ERROR_C := DWORD#0;
//
// 		X.UCB.D_MODE := 99;
// 		UCB(DATA:=X.UCB); (* clear buffer *)
//
// 		URL_DATA:=STRING_TO_URL(STR:=URL,DEFAULT_PROTOCOL:='',DEFAULT_PATH:=''); (* split URL *)
// 		sep_char := CHR_TO_STRING(SEP);
// 		url_query := URL_DATA.QUERY;
// 		step_1 := 30;
//
// 		(* ---------------- Debug-Message -----------------------*)
// 		(*IF _debug_enable THEN
// 			LOG_CL.NEW_MSG := 'FILE_RRD1 - Start: DATE [~2]';
// 			LOG_CL.PRINTF[2] := DT_TO_STRING(DTI);
// 			LOG_MSG();
// 		END_IF;*)
// 		(* -----------------------------------------------------------------*)
//
// 	END_IF;
//
// 30:	(* process LOG trigger *)
// 	trig_tmp := (TRIG_M AND NOT trig_m_last) OR trig_auto OR X.ADD_DATA_REQ;
//
// 	IF ENABLE = FALSE THEN (* ENABLE = 0 -> Log Stop *)
// 		X.ADD_COM := 00;
// 		step_1 := 00;
//
// 		(* ---------------- Debug-Message -----------------------*)
// 		(*IF _debug_enable THEN
// 			LOG_CL.NEW_MSG := 'FILE_RRD1 - Stop: DATE [~2]';
// 			LOG_CL.PRINTF[2] := DT_TO_STRING(DTI);
// 			LOG_MSG();
// 		END_IF;*)
// 		(* -----------------------------------------------------------------*)
//
// 	ELSIF ENABLE THEN
// 		IF trig_tmp OR trig_stored THEN (* manual, automatic or external trigger *)
// 			trig_stored := FALSE;
// 			X.ADD_COM := 03; (* ADD DATA *)
// 			(* ---------------- Debug-Message -----------------------*)
// 			(*IF _debug_enable THEN
// 				LOG_CL.NEW_MSG := 'FILE_RRD1 - Trig: DATE [~2]';
// 				LOG_CL.PRINTF[2] := DT_TO_STRING(DTI);
// 				LOG_MSG();
// 			END_IF;*)
// 			(* -----------------------------------------------------------------*)
// 		ELSE
// 			X.ADD_COM := 04;	(* ADD DATA REQ *)
// 		END_IF;
// 	END_IF;
//
// END_CASE;
// X.ADD_DATA_REQ := FALSE; (* reset external request *)
//
// (* ##################################### *)
//
// CASE step_2 OF
//
// 00:	IF X.UCB.BUF_DATA_LOST > UDINT#0 THEN
// 		ERROR_C := DWORD#2; (* error: buffer overflow - reduce amount of data *)
// 		ERROR_T := BYTE#6; 	(* Type: Buffer *)
// 		step_2 := 100;
// 	ELSIF X.UCB.BUF_USED_MAX > USINT#90 THEN
// 		ERROR_C := DWORD#1; (* warning: buffer utilization > 90% *)
// 		ERROR_T := BYTE#6;	(* Type: Buffer *)
// 	END_IF;
//
// 	IF X.UCB.BUF_COUNT >= USINT_TO_INT(X.ID_MAX) THEN (* enough entries available *)
// 		URL_DATA.QUERY := url_query; (* restore original query *)
// 		n := 1;
// 		WHILE n <= USINT_TO_INT(X.ID_MAX) DO
// 			X.UCB.D_MODE := 12; (* read and delete element *)
// 			UCB(DATA:=X.UCB);
// 			IF n < USINT_TO_INT(X.ID_MAX) THEN (* add separator *)
// 				X.UCB.D_STRING := CONCAT(X.UCB.D_STRING,sep_char);
// 			END_IF;
// 			IF LEN(X.UCB.D_STRING) + LEN(URL_DATA.QUERY) <= STRING_LENGTH THEN
// 				URL_DATA.QUERY := CONCAT(URL_DATA.QUERY,X.UCB.D_STRING); (* append LOG data to query *)
// 				step_2 := 40;
// 			ELSE
// 				ERROR_T := BYTE#4; (* LOG data cannot be packed into the URL *)
// 				ERROR_C := DWORD#1;
// 				step_2 := 100;
// 			END_IF;
// 			n := n + 1;
// 		END_WHILE;;
// 	END_IF;
//
// 40:	IF DNS_CLIENT.DONE THEN
// 		step_2 := 60;
// 	ELSIF (DNS_CLIENT.ERROR > DWORD#0) THEN
// 		ERROR_C := DNS_CLIENT.ERROR; (* error handling *)
// 		ERROR_T := BYTE#1;
// 		step_2 := 100;
// 	END_IF;
//
// 60:	IF HTTP_GET.DONE THEN
// 		n := UINT_TO_INT(HTTP_GET.BODY_START);
// 		IF R_BUF.BUFFER[n] <> BYTE#48 THEN (* ASCII '0' *)
// 			ERROR_C := DWORD#1;
// 			ERROR_T := BYTE#3;
// 		END_IF;
// 		step_2 := 100;
//
// 	ELSIF HTTP_GET.ERROR > DWORD#0 THEN (* error handling *)
// 		ERROR_C := HTTP_GET.ERROR;
// 		ERROR_T := BYTE#2;
// 		step_2 := 100;
// 	END_IF;
//
// 100:	IF (NOT HTTP_GET.DONE) THEN (* UNLOCK HTTP DATA *)
// 		step_2 := SEL(ERROR_T = BYTE#0, 120,0);
// 	END_IF;
//
// 120:	IF NOT ENABLE THEN
// 		step_2 := 0;
// 	END_IF;
//
// END_CASE;
//
// HTTP_GET(IP_C:=IP_C,S_BUF:=S_BUF,R_BUF:=R_BUF,IP4:=DNS_CLIENT.IP4,GET:=step_2=60,MODE:=2,UNLOCK_BUF:=step_2=100,URL_DATA:=URL_DATA); (* HTTP_GET *)
// DNS_CLIENT(IP_C:=IP_C, S_BUF:=S_BUF, R_BUF:=R_BUF, DOMAIN:=URL_DATA.DOMAIN, IP4_DNS:= DNS_IP4, ACTIVATE:=step_2=40); (* DNS-Client *)
// IPC(IP:= 0, PORT:= 0 , TIME_OUT:= TIMEOUT, IP_C:= IP_C, S_BUF:= S_BUF, R_BUF:= R_BUF); (* IP_CONTROL *)
//
// trig_m_last := TRIG_M;
// END_FUNCTION_BLOCK

// Commented out for beedance: it uses UNI_CIRCULAR_BUFFER, which is commented out.
// FUNCTION_BLOCK DLOG_STRING
// VAR_IN_OUT
// 	X : DLOG_DATA;
// END_VAR
// VAR_INPUT
// 	STR : STRING;
// 	COLUMN : STRING(40);
// END_VAR
// VAR_OUTPUT
// END_VAR
// VAR
// 	UCB : UNI_CIRCULAR_BUFFER;
// 	id : WORD;
// 	str_last : STRING;
// END_VAR
//
// CASE x.ADD_COM OF
//
// 01:	(* ADD INFO *)
// 	X.ID_MAX := X.ID_MAX + USINT#1;
// 	id := WORD#16#0101; (* source type STRING, target type STRING *)
// 02:	(* ADD HEADER *)
// 	X.UCB.D_STRING := COLUMN;
// 	X.UCB.D_HEAD := id;
// 	X.UCB.D_MODE := 1;
// 	UCB(DATA:=X.UCB); (* enter data *)
// 03:	(* ADD DATA *)
// 	X.UCB.D_STRING := str_last;
// 	X.UCB.D_HEAD := id;
// 	X.UCB.D_MODE := 1;
// 	UCB(DATA:=X.UCB); (* enter data *)
// END_CASE;
// str_last := STR;
// END_FUNCTION_BLOCK

// Commented out for beedance: it uses CODE, which is commented out.
// FUNCTION_BLOCK DNS_CLIENT
// VAR_IN_OUT
// 	IP_C : IP_C; (* IP_Control management structure *)
// 	S_BUF : NETWORK_BUFFER;
// 	R_BUF : NETWORK_BUFFER;
// END_VAR
// VAR_INPUT
// 	ACTIVATE : BOOL;
// 	DOMAIN : STRING;
// 	IP4_DNS : DWORD;
// END_VAR
// VAR_OUTPUT
// 	IP4 : DWORD;
// 	DONE : BOOL;
// 	ERROR : DWORD;
// END_VAR
// VAR
// 	IP_FIFO : IP_FIFO;
// 	ip_state : BYTE;
// 	ip_id : BYTE;
// 	i : INT;
// 	state : INT;
// 	domain_copy : STRING;
// 	activate_last : BOOL;
// 	url_length : INT;
// 	char : BYTE;
// 	char_count : INT;
// 	tid : BYTE;
// 	anc : INT;
// 	x : BYTE;
// 	rr_stop : BOOL;
// 	ttl_last : DWORD;
// 	ttl_tmp : DWORD;
//
// 	(*LOG_MSG : LOG_MSG;
// 	_debug_enable : BOOL := TRUE;*)
//
// END_VAR
//
// (* Domain Name System (query) *)
//
// CASE state OF
//
// 00:	IF ACTIVATE AND NOT activate_last THEN (* wait for rising edge on GET *)
// 		DONE := FALSE;
// 		ERROR := DWORD#0;
// 		state := 5;
// 	END_IF;
//
// 05:	IP4 := IP4_DECODE(str:=DOMAIN); (* check whether domain is already an IP4 address *)
// 	IF IP4 > DWORD#00 THEN
// 		DONE := TRUE;
// 		state := 0;
//         		(*####################  DEBUG-MESSAGE  ###################################*)
//         		(*IF _debug_enable THEN
//             		LOG_CL.NEW_MSG := 'DNS: S05 IP4 ~1';
//             		LOG_CL.PRINTF[1]  := DOMAIN;
//             		LOG_MSG();
//         		END_IF;*)
//         		(*########################################################################*)
// 	ELSE
// 		ip_state := BYTE#1;
// 		ttl_last := DWORD#0;
// 		domain_copy := DOMAIN; (* save DOMAIN string *)
// 		state := 10;
//         		(*####################  DEBUG-MESSAGE  ###################################*)
//         		(*IF _debug_enable THEN
//             		LOG_CL.NEW_MSG := 'DNS: S05 START';
//             		LOG_MSG();
//         		END_IF;*)
//         		(*########################################################################*)
// 	END_IF;
//
// 10:	IF ip_state = BYTE#3 THEN (* register with IP_Control *)
// 		url_length := LEN(domain_copy);
// 		char_count := 17 + url_length; (* initialize send buffer *)
// 		FOR i := 0 TO char_count DO
// 			S_BUF.BUFFER[i] := BYTE#00;
// 		END_FOR;
// 		tid := UINT_TO_BYTE(BYTE_TO_UINT(tid) + UINT#1);
// 		S_BUF.BUFFER[01] := tid; (* Transaction ID lowbyte *)
// 		S_BUF.BUFFER[02] := BYTE#16#01; (* Flags: highbyte *)
// 		S_BUF.BUFFER[05] := BYTE#16#01; (* Questions: lowbyte *)
// 		i := url_length + 12;	(* process the server name from back to front *)
// 		char_count := 0;
// 		WHILE i > 12 DO
// 			char := CODE(STR:=domain_copy,POS:=i - 12);
// 			IF char = BYTE#46 THEN (* check for main/sub domain name separator "." *)
// 				S_BUF.BUFFER[i] := INT_TO_BYTE(char_count); (* instead of the separator "." the length of the detected main/sub domain name is entered *)
// 				char_count := 0;
// 			ELSE
// 				S_BUF.BUFFER[i] := char; (* enter char into buffer *)
// 				char_count := char_count + 1; (* count number of chars *)
// 			END_IF;
// 			i := i - 1;
// 		END_WHILE;
// 		S_BUF.BUFFER[i] := INT_TO_BYTE(char_count); (* enter the length of the leftmost (first) domain name *)
// 		i := url_length + 15; (* position after the server name *)
// 		S_BUF.BUFFER[i] := BYTE#01; (* Type: A Hostaddress lowbyte *)
// 		i := i + 2;
// 		S_BUF.BUFFER[i] := BYTE#01; (* Class: IN lowbyte *)
// 		i := i + 1;
// 		(* set up IP data traffic *)
// 		IP_C.C_PORT := WORD#53; (* enter port number *)
// 		IP_C.C_IP := IP4_DNS; (* enter IP *)
// 		IP_C.C_MODE := BYTE#1; (* Mode: UDP+ACTIVE+PORT+IP *)
// 		IP_C.C_ENABLE := TRUE; (* enable connection setup *)
// 		IP_C.TIME_RESET := TRUE; (* reset timeout monitoring *)
// 		IP_C.R_OBSERVE  := TRUE; (* monitor data reception *)
// 		S_BUF.SIZE := INT_TO_UINT(i); (* enter send length *)
// 		R_BUF.SIZE := UINT#0; (* reset receive length *)
// 		state := 30;
//
//         		(*####################  DEBUG-MESSAGE  ###################################*)
//         		(*IF _debug_enable THEN
//             		LOG_CL.NEW_MSG := 'DNS: S10 SEND';
//             		LOG_MSG();
//         		END_IF;*)
//         		(*########################################################################*)
// 	END_IF;
//
// 30:	IF IP_C.ERROR <> DWORD#00 THEN
// 		ERROR := IP_C.ERROR;
// 		state := 99;
//         		(*####################  DEBUG-MESSAGE  ###################################*)
//         		(*IF _debug_enable THEN
//             		LOG_CL.NEW_MSG := 'DNS: S30 ERROR ~1';
//             		LOG_CL.PRINTF[1]  := DWORD_TO_STRING(ERROR);
//             		LOG_MSG();
//         		END_IF;*)
//         		(*########################################################################*)
//
// 	ELSIF (S_BUF.SIZE = UINT#0) AND (tid = R_BUF.BUFFER[1]) AND (R_BUF.SIZE >= INT_TO_UINT(34 + url_length)) THEN	(* check whether the response telegram has the correct transaction ID and minimum length *)
// 		ERROR := BYTE_TO_DWORD(R_BUF.BUFFER[3] AND BYTE#2#0000_1111); (* check return code of the flags. 4 bits *)
// 		IF ERROR = DWORD#00 THEN
// 			anc := R_BUF.BUFFER[7]; (* number of answer RRs *)
// 			IP_C.R_OBSERVE := FALSE; (* monitor data reception *)
// 			state := 40;
// 		ELSE
// 			state := 99;
// 		END_IF;
// 	END_IF;
//
// 40:	IF anc > 0 THEN
// 		anc := anc - 1;
// 		WHILE i < R_BUF.SIZE DO
// 			x := R_BUF.BUFFER[i];
// 			IF rr_stop = FALSE THEN
// 				IF x > BYTE#63 THEN (* pointer to name *)
// 					i := i + 1;
// 					rr_stop := TRUE;
// 				ELSIF x= BYTE#0 THEN (* end of name *)
// 					rr_stop := TRUE;
// 				ELSE
// 					i := i + x; (* names *)
// 				END_IF;
// 				i := i + 1;
// 			ELSE
// 				rr_stop := FALSE;
// 				IF R_BUF.BUFFER[i+1] = BYTE#1 AND R_BUF.BUFFER[i+3] = BYTE#1 THEN (* Type A / Class IN *)
// 					i := i + 4;
// 					ttl_tmp := DWORD_OF_BYTE(R_BUF.BUFFER[i],R_BUF.BUFFER[i+1],R_BUF.BUFFER[i+2],R_BUF.BUFFER[i+3]); (* Time to live *)
// 					i := i + 6;
// 					IF ttl_tmp >= ttl_last THEN (* TTL is longer *)
// 						ttl_last := ttl_tmp;
// 						IP4 := DWORD_OF_BYTE(R_BUF.BUFFER[i],R_BUF.BUFFER[i+1],R_BUF.BUFFER[i+2],R_BUF.BUFFER[i+3]); (* IP address *)
// 					END_IF;
// 					i := i + 4;
// 				ELSE
// 					i := i + 9;
// 					i := i + R_BUF.BUFFER[i] + 1; (* offset to next block *)
// 				END_IF;
// 				EXIT;
// 			END_IF;
// 		END_WHILE;
// 	ELSE
// 		IF IP4 > DWORD#0 THEN (* valid RR with IP found *)
// 			DONE := TRUE;
//             		(*####################  DEBUG-MESSAGE  ###################################*)
//             		(*IF _debug_enable THEN
//                 			LOG_CL.NEW_MSG := 'DNS: S40 OK';
//                 			LOG_MSG();
//             		END_IF;*)
//             		(*########################################################################*)
// 		ELSE
// 			ERROR := DWORD#255; (* data faulty - no IP address present *)
// 		END_IF;
// 		state := 99;
// 	END_IF;
//
// 99:	R_BUF.SIZE := UINT#0; (* reset receive length *)
// 	ip_state := BYTE#4; (* unregister *)
// 	state := 00;
//
// END_CASE;
//
// activate_last := ACTIVATE; (* save last status for edge detection *)
// IP_FIFO(FIFO:=IP_C.FIFO,STATE:=ip_state,ID:=ip_id); (* IP_FIFO *)
//
// (*----------------------------------------------------------------------------------------------------------------*)
// (* Flags: 0x0100 (Standard query)                                                                                            *)
// (* 0... .... .... .... = Response: Message is a query                                                                   *)
// (* .000 0... ....  = Opcode: Standard query (0)                                                                          *)
// (* .... ..0. .... .... = Truncated: Message is not truncated                                                          *)
// (* .... ...1 .... .... = Recursion desired: Do query recursively                                                    *)
// (* .... .... .0.. .... = Z: reserved (0)                                                                                                  *)
// (* .... .... ...0 .... = Non-authenticated data OK: Non-authenticated data is unacceptable *)
// (*-----------------------------------------------------------------------------------------------------------------*)
//
// (*      0  1  2  3  4  5  6  7  8  9  0  1  2  3  4  5  *)
// (*    +--+--+--+--+--+--+--+--+--+--+--+--+--+--+--+--+ *)
// (*    |                      ID                       | idx: 0/1   *)
// (*    +--+--+--+--+--+--+--+--+--+--+--+--+--+--+--+--+ *)
// (*    |QR|   Opcode  |AA|TC|RD|RA|   Z    |   RCODE   | idx: 2/3   *)
// (*    +--+--+--+--+--+--+--+--+--+--+--+--+--+--+--+--+ *)
// (*    |                    QDCOUNT                    | idx: 4/5   *)
// (*    +--+--+--+--+--+--+--+--+--+--+--+--+--+--+--+--+ *)
// (*    |                    ANCOUNT                    | idx: 6/7   *)
// (*    +--+--+--+--+--+--+--+--+--+--+--+--+--+--+--+--+ *)
// (*    |                    NSCOUNT                    | idx: 8/9   *)
// (*    +--+--+--+--+--+--+--+--+--+--+--+--+--+--+--+--+ *)
// (*    |                    ARCOUNT                    | idx: 10/11 *)
// (*    +--+--+--+--+--+--+--+--+--+--+--+--+--+--+--+--+ *)
//
// (*
// Errorcodes  Description	References
// 000	No error. 		 	The request completed successfully.
// 001	Format error. 		The name server was unable to interpret the query.
// 002	Server failure.  	The name server was unable to process this query due to a problem with the name server.
// 003	Name Error. 	 	Meaningful only for responses from an authoritative name server, this code signifies that the domain name referenced in the query does not exist.
// 004	Not Implemented. 	The name server does not support the requested kind of query.
// 005	Refused. 			The name server refuses to perform the specified operation for policy reasons.
//   						 For example, a name server may not wish to provide the information to the particular requester, or a name server may not wish to perform a particular operation (e.g., zone transfer) for particular data.
// 006	YXDomain.			Name Exists when it should not.
// 007	YXRRSet. RR			Set Exists when it should not.
// 008	NXRRSet. RR			Set that should exist does not.
// 009	NotAuth.			Server Not Authoritative for zone.
// 010	NotZone,			Name not contained in zone.
// 255	Timeout				No Response
//
// example of a DNS request for google.at
// a request with 3 answer blocks
//
// Domain Name System (response)
// [Request In: 3]
// [Time: 0.027533000 seconds]
// Transaction ID: 0x5e1a
// Flags: 0x8180 (Standard query response, No error)
// 1... .... .... .... = Response: Message is a response
// .000 0... .... .... = Opcode: Standard query (0)
// .... .0.. .... .... = Authoritative: Server is not an authority for domain
// .... ..0. .... .... = Truncated: Message is not truncated
// .... ...1 .... .... = Recursion desired: Do query recursively
// .... .... 1... .... = Recursion available: Server can do recursive queries
// .... .... .0.. .... = Z: reserved (0)
// .... .... ..0. .... = Answer authenticated: Answer/authority portion was not authenticated
// .... .... .... 0000 = Reply code: No error (0)
// Questions: 1
// Answer RRs: 3
// Authority RRs: 0
// Additional RRs: 0
//
// Queries
// google.at: type A, class IN
// Name: google.at
// Type: A (Host address)
// Class: IN (0x0001)
//
// Answers
// google.at: type A, class IN, addr 72.14.221.104
// Name: google.at
// Type: A (Host address)
// Class: IN (0x0001)
// Time to live: 19 minutes, 9 seconds
// Data length: 4
// Addr: 72.14.221.104
//
// google.at: type A, class IN, addr 66.249.93.104
// Name: google.at
// Type: A (Host address)
// Class: IN (0x0001)
// Time to live: 19 minutes, 9 seconds
// Data length: 4
// Addr: 66.249.93.104
//
// google.at: type A, class IN, addr 216.239.59.104
// Name: google.at
// Type: A (Host address)
// Class: IN (0x0001)
// Time to live: 19 minutes, 9 seconds
// Data length: 4
// Addr: 216.239.59.104
// *)
// END_FUNCTION_BLOCK

// Commented out for beedance: it uses BUFFER_TO_STRING, which is commented out.
// FUNCTION_BLOCK DNS_DYN
// VAR_IN_OUT
// 	IP_C : IP_C; (* IP_Control management structure *)
// 	S_BUF : NETWORK_BUFFER;
// 	R_BUF : NETWORK_BUFFER;
// END_VAR
// VAR_INPUT
// 	ENABLE : BOOL;
// 	UPDATE : BOOL;
// 	T_UPDATE : TIME := T#1h;
// 	MODE : BYTE;
// 	HOSTNAME : STRING(30);
// 	USERNAME : STRING(20);
// 	PASSWORD : STRING(20);
// 	IP4 : DWORD;
// END_VAR
// VAR_OUTPUT
// 	BUSY : BOOL;
// 	DONE : BOOL;
// 	ERROR_C : DWORD;
// 	ERROR_T : BYTE;
// END_VAR
// VAR
// 	DNS_CLIENT : DNS_CLIENT;
// 	HTTP_GET : HTTP_GET;
// 	BASE64_ENCODE_STR : BASE64_ENCODE_STR;
// 	URL_DATA : url;
// 	update_last : BOOL;
// 	state : INT;
// 	base64_done : BOOL;
// 	s1 : STRING(144);
// 	s2 : STRING(192);
// 	w : TON;
// END_VAR
//
// CASE state OF
//
// 00:	IF ENABLE AND ((UPDATE AND NOT update_last) OR w.Q) THEN
// 		state := 20;
// 		DONE := FALSE;
// 		BUSY := TRUE;
// 		ERROR_C := DWORD#0;
// 		ERROR_T := BYTE#0;
//
// 		IF MODE = 0 THEN (* dyndns.org *)
// 			s2 := CONCAT('http://members.dyndns.org/nic/update?hostname=',HOSTNAME);
// 		ELSE (* selfhost.de *)
// 			s2 := 'http://carol.selfhost.de/nic/update?hostname=1';
// 		END_IF;
// 		IF IP4 > 0 THEN (* use configured IP *)
// 			s1 := CONCAT('&myip=',IP4_TO_STRING(IP4));
// 			s2 := CONCAT(s2,s1);
// 		END_IF;
// 		URL_DATA:=STRING_TO_URL(STR:=s2, DEFAULT_PROTOCOL:='', DEFAULT_PATH:=''); (* URL for DNS AND HTTP-GET *)
// 		s1 := CONCAT(USERNAME,':');
// 		s1 := CONCAT(s1,PASSWORD); (* BASE64 Encode Text *)
// 	END_IF;
//
// 20:	IF DNS_CLIENT.DONE THEN (* DNS_CLIENT *)
// 			state := 40;
// 	ELSIF (DNS_CLIENT.ERROR > DWORD#00) THEN (* error handling *)
// 		ERROR_C := DNS_CLIENT.ERROR;
// 		ERROR_T := BYTE#01;
// 		BUSY := FALSE;
// 		state := 0;
// 	END_IF;
//
// 40: IF base64_done THEN (* BASE64 encode finished? *)
// 		s1 := CONCAT('Authorization: Basic ',s2);
// 		s1 := CONCAT(s1,'$0D$0AUser-Agent: x$0D$0A');
// 		URL_DATA.HEADER := s1;
// 		state := 60;
// 	END_IF;
//
// 60:	IF HTTP_GET.DONE THEN
// 		state := 0;
// 		BUSY := FALSE;
// 		DONE := TRUE;
//
// 		(* !! Codes !!
// 		Successful Updates: 		good , nchg
// 		Update Syntax Errors:		badsys , badagent
// 		Account-Related Errors:		badauth , !donator
// 		Hostname-Related Errors:	notfqdn , nohost , !yours , numhost , abuse
// 		Server Error Conditions:	dnserr , 911
// 		*)
// 		s2 := BUFFER_TO_STRING(PT:=REF(R_BUF.BUFFER),SIZE:=SIZEOF(R_BUF.BUFFER),START:=HTTP_GET.BODY_START + 3,STOP:=HTTP_GET.BODY_STOP - 7);
// 		IF FIND(s2,'good') = 0 THEN
// 			IF FIND(s2,'nochg') = 0 THEN
// 				ERROR_C := DWORD#1;
// 				ERROR_T := BYTE#03;
// 				DONE := FALSE;
// 			END_IF;
// 		END_IF;
// 	ELSIF (HTTP_GET.ERROR > DWORD#00) THEN (* error handling *)
// 		ERROR_C := HTTP_GET.ERROR;
// 		ERROR_T := BYTE#02;
// 		BUSY := FALSE;
// 		state := 0;
// 	END_IF;
//
// END_CASE;
//
// DNS_CLIENT(IP_C:=IP_C,	S_BUF:=S_BUF, R_BUF:=R_BUF,DOMAIN:=URL_DATA.DOMAIN, IP4_DNS:=0, ACTIVATE:=state=20); (* DNS_CLIENT *)
// HTTP_GET( IP_C:=IP_C, S_BUF:=S_BUF, R_BUF:=R_BUF, IP4:=DNS_CLIENT.IP4, GET:=state=60, MODE:=2, UNLOCK_BUF:=state<>60,URL_DATA:=URL_DATA); (* HTTP_GET *)
// BASE64_ENCODE_STR( RUN:=state=40, STR1:=s1, STR2:=s2, DONE=>base64_done); (* BASE64 Encode *)
//
// IF T_UPDATE > T#0ms THEN w(IN:=state=0, PT:=T_UPDATE); END_IF;
// update_last := UPDATE;
// END_FUNCTION_BLOCK
